# B&R Automation Studio project MotionTestBenchMaster (part 13)

#### ETHIP_COM.st - ETHIP COM Code
```iecst
(************************************************************************************************************************)
(* COPYRIGHT -- Sidel S.p.a.                                                                                            *)
(************************************************************************************************************************)
(* Library:				ETHIP_COM																						*)
(* Author:				Andrea.Cortesi																					*)
(* Site:				Sidel - Parma - Product Care IO																	*)
(* Created:				August 26, 2015																					*)
(* Description:			This Library manage a communication based on ethernet IP Protocol between plc B&R configurated	*)
(*						like a SLAVE and another plc configurated like a MASTER. Connection is openinig only if partner	*)
(*						give positive response at comand ping. In case of timeout connection (5000 ms is default value)	*)
(*						the library close connection, try again to ping partner and if there is no answer generate fault*)
(*						communication. Fault is generate also if there is an error inside Data Object configuration.	*)
(* Restriction:			Call in Fast Task at 30 ms or less.Only one connection can be activated because plc B&R in SLAVE*)
(*						Plc B&R can not be SLAVE of two MASTER at same time!!! Is not possible open two connections like*)
(*						SLAVE concurrently on the same IFx eth port. However is possible open two connections like SLAVE*)
(*						Sconcurrently on two different eth port (ex:IF2 and IF3) with two different IP address class	*)
(* Important Note:		This library open/close connection (with memory release) also in case of program download made	*)
(*						in Copy Mode or Overload Mode.For correct management of Overload Mode is necessaary call istance*)
(*						of ETHIP library with Enable at FALSE inside Exit Transiction of function block in which ETHIP	*)
(*						library istance is called.																		*)
(*----------------------------------------------------------------------------------------------------------------------*)
(* Version History:		v.4.00.0 Date 2015-09-12  Andrea.Cortesi														*)
(* Version History:		v.4.00.1 Date 2017-08-20  Roberto.Bonato														*)
(*																														*)
(*----------------------------------------------------------------------------------------------------------------------*)
(* Development Tool:	B&R Automation Studio V3.0.90.27 SP09															*)
(* Compiler GCC:		V2.95.3; V4.1.1; V4.1.2																			*)
(*----------------------------------------------------------------------------------------------------------------------*)
(* Dependencies:		AsEthIP,AsICMP,AsString,Runtime,Standard														*)
(************************************************************************************************************************)

FUNCTION_BLOCK ETHIP_COM
   (* PING Partner before Communication Initialisation *)
	IF (Enable AND NOT(Ping_Ok) AND NOT(Error)) THEN
		PING_Partner.enable		:= TRUE;
		PING_Partner.pHost		:= ADR(IP_Address_Partner);
		PING_Partner.timeout	:= 500;
		PING_Partner();

		Step_Msg_Active      := 'ETHIP PING';
		Status               := PING_Partner.status;
		ETHIP_COM_Error;	(* Call action ETHIP_COM_Error *)

		CASE PING_Partner.status OF
			0:		(* No Error *)
				Ping_Ok	:= TRUE;

			32750,	(* No response sent by station within the specified timeout *)
			32751,	(* The specified IP address (SG4: name also) could not be resolved *)
			32752,	(* Resource problem in system. Could not create new sockets *)
			65535:	(* No Error - Function block still operating, continue calling *)
				Ping_Ok	:= FALSE;
			ELSE	(* Error not management *)
				Ping_Ok	:= FALSE;
		END_CASE
	END_IF

	(* ETHIP Communication Initialisation *)
	IF ComInit THEN	(* If the communication initialisation is requested then... *)
		ETHIP_Init.enable	:= TRUE;				(* Enabled *)
		ETHIP_Init.pconfig	:= Config_DataObject;	(* Name of the "communication configuration" data object *)
		ETHIP_Init();								(* Call of the "EIPInit" function *)

		Handle_Init			:= ETHIP_Init.handle;	(* The handle returned by the EIPInit Function and is reused by the EIPCyclic AND EIPExit functions *)

		Step_Msg_Active		:= 'ETHIP INIT';
		Status				:= ETHIP_Init.status;
		ETHIP_COM_Error;							(* Call action ETHIP_COM_Error *)

		(* ETHIP Status Init *)
		CASE ETHIP_Init.status OF
			0:		(* No Error *)
				ComInit		:= FALSE;		(* Reset the communication init request *)
				ComStart	:= TRUE;		(* Set the communication activation request *)

			32051,	(* Out of memory. The library cannot be executed *)
			32052,	(* Configuration data object error *)
			32053,	(* Illegal input parameters connected to the FBK. *)
			32054:	(* The Ethernet interface doesn't exist or returns an error. Check the #OWNINTERFACE entry in the configuration data object.*)
				ComInit		:= FALSE;		(* Reset the communication init request *)
				ComStart	:= FALSE;		(* Reset the communication activation request *)
				ComExit		:= TRUE;		(* Set the communication exit request *)

			65534:	(* The FBK was called with enable = 0.*)

			65535:	(* No Error - Function block still operating, continue calling *)

			ELSE	(* Error not management *)
				ComInit		:= FALSE;		(* Reset the communication init request *)
				ComStart	:= FALSE;		(* Reset the communication activation request *)
				ComExit		:= FALSE;		(* Reset the communication exit request *)
		END_CASE
	END_IF

	(* ETHIP Communication Cyclic *)
	IF ComStart THEN		(* If communication activation is requested then... *)
		ETHIP_Cyclic.enable	:= TRUE;		(* Enabled *)
		ETHIP_Cyclic.handle	:= Handle_Init;	(* Handle received from the EIPInit function *)
		ETHIP_Cyclic();						(* Call of the "EIPcyclic" function *)

		Step_Msg_Active		:= 'ETHIP CYCLIC';
		Status				:= ETHIP_Cyclic.status;
		ETHIP_COM_Error;					(* Call action ETHIP_COM_Error *)
	END_IF

	(* ETHIP Status Cyclic *)
	CASE ETHIP_Cyclic.status OF
		0:		(* No Error *)

		32051,	(* Out of memory. The library cannot be executed *)
		32052,	(* Configuration data object error *)
		32053,	(* Illegal input parameters connected to the FBK. *)
		32054:	(* The Ethernet interface doesn't exist or returns an error. Check the #OWNINTERFACE entry in the configuration data object.*)
			ComStart	:= FALSE;		(* Reset the communication activation request *)
			ComExit		:= TRUE;		(* Set the communication exit request *)

		65534:	(* The FBK was called with enable = 0.*)

		65535:	(* No Error - Function block still operating, continue calling *)

		ELSE	(* Error not management *)
			ComInit		:= FALSE;	(* Reset the Communication init request *)
			ComStart	:= FALSE;	(* Reset the communication activation request *)
			ComExit		:= FALSE;	(* Reset the communication exit request *)
	END_CASE

	(* Force ETHIP Communication Exit if Enable Not Active *)
	IF (NOT(Enable) AND (ComStart OR ComInit)) THEN
		ComInit		:= FALSE;	(* Reset the communication init request *)
		ComStart	:= FALSE;	(* Reset the communication activation request *)
		ComExit		:= TRUE;	(* Set the communication exit request *)
	END_IF

	(* ETHIP Communication Exit *)
	IF ComExit THEN	(* If communication exit is requested then... *)
		ComInit		:= FALSE;		(* Reset the communication init request *)
		ComStart	:= FALSE;		(* Reset the communication activation request *)

		ETHIP_Exit.enable	:= TRUE;		(* Enabled *)
		ETHIP_Exit.handle	:= Handle_Init;	(* Handle received from the EIPInit function *)
		ETHIP_Exit();						(* Call of the "EIPExit" function *)

		Step_Msg_Active		:= 'ETHIP EXIT';
		Status				:= ETHIP_Exit.status;
		ETHIP_COM_Error;					(* Call action ETHIP_COM_Error *)
	END_IF

	(* ETHIP Status Exit *)
	CASE ETHIP_Exit.status OF
		0:		(* No Error *)

		32051,	(* Out of memory. The library cannot be executed *)
		32052,	(* Configuration data object error *)
		32053,	(* Illegal input parameters connected to the FBK. *)
		32054:	(* The Ethernet interface doesn't exist or returns an error. Check the #OWNINTERFACE entry in the configuration data object.*)
			ComInit		:= FALSE;	(* Reset the communication init request *)
			ComStart	:= FALSE;	(* Reset the communication activation request *)
			ComExit		:= FALSE;	(* Reset the communication exit request *)

		65534:	(* The FBK was called with enable = 0. *)

		65535:	(* No Error - Function block still operating, continue calling *)

		ELSE	(* Error not management *)
			ComInit		:= FALSE;	(* Reset the communication init request *)
			ComStart	:= FALSE;	(* Reset the communication activation request *)
			ComExit		:= FALSE;	(* Reset the communication exit request *)
	END_CASE

	// Check if ETHIP Communication Exit is Ended
	IF (ComExit AND (ETHIP_Exit.status = 0)) THEN
		ComInit		:= FALSE;		(* Reset the communication init request *)
		ComStart	:= FALSE;		(* Reset the communication activation request *)
		ComExit		:= FALSE;		(* Reset the communication exit request *)
	END_IF

	// Check Presence Status Error in ETHIP Init and ETHIP Cyclic
	IF ((ETHIP_Init.status = 0) OR (ETHIP_Init.status = 65335)) AND ((ETHIP_Cyclic.status = 0) OR (ETHIP_Cyclic.status = 65335)) THEN
		Error_Internal	:= FALSE;	(* Reset Error in ETHIP function *)
	ELSE
		IF Ping_Ok THEN
			Error_Internal	:= TRUE;	(* Set Error in ETHIP function *)
		ELSE
			Error_Internal	:= FALSE;	(* Reset Error in ETHIP function *)
		END_IF
	END_IF

	// Set Communication Exit if Ping Not Ok or Fault Communication
	IF (ComStart AND (EDGEPOS(Error) OR EDGENEG(Ping_Ok))) THEN
		IF ConnectionAttempt > 10 THEN
			ComInit		:= FALSE;		(* Reset the communication init request *)
			ComStart	:= FALSE;		(* Reset the communication activation request *)
			ComExit		:= TRUE;		(* Set the communication exit request *)
			ConnectionAttempt := 0;
		ELSE
			ConnectionAttempt	:= ConnectionAttempt + 1;
			Error := FALSE;
		END_IF
	ELSIF (ComStart AND EDGE(Alive_Bit_From_Partner)) THEN
		ConnectionAttempt := 0;
	END_IF

	// Initializatin Communication
	IF (Enable AND NOT(ComInit) AND NOT(ComStart) AND NOT(ComExit) AND Ping_Ok AND NOT(Error)) THEN
		ComInit		:= TRUE;		(* Set the communication init request *)
		ComStart	:= FALSE;		(* Reset the communication activation request *)
		ComExit		:= FALSE;		(* Reset the communication exit request *)
	END_IF

	// Check TimeOut Value
	IF (TimeOut_Value = 0) THEN
		TimeOut_Value	:= 5000;
	ELSIF (TimeOut_Value < 3000) THEN
		TimeOut_Value	:= 3000;
	END_IF

	// Check Alive Bit Receive from Partner
	IF Enable THEN
		Timer_CommTimeOut(
		IN	:= NOT EDGE(Alive_Bit_From_Partner) AND Timer_StartComDelay.Q,
		PT	:= UINT_TO_TIME(TimeOut_Value)
		);

		Timer_StartComDelay(
		IN	:= TRUE,
		PT	:= UINT_TO_TIME(TimeOut_Value)
		);
	ELSE
		Timer_CommTimeOut(
		IN	:= FALSE,
		PT	:= UINT_TO_TIME(TimeOut_Value)
		);

		Timer_StartComDelay(
		IN	:= FALSE,
		PT	:= UINT_TO_TIME(TimeOut_Value)
		);
	END_IF

	// TimeOut Error Communication
	IF ((NOT(Ping_Ok) AND Timer_CommTimeOut.Q) OR Error_Internal) THEN
		Timer_CommTimeOut.IN	:= FALSE;
		Timer_StartComDelay.IN	:= FALSE;
		Error					:= TRUE;
	END_IF

	// Try again to Ping Partner in case of TimeOut Error Communication
	IF (Ping_Ok AND Timer_CommTimeOut.Q AND NOT(Error)) THEN
		Timer_CommTimeOut.IN	:= FALSE;
		Timer_StartComDelay.IN	:= FALSE;
		Ping_Ok					:= FALSE;
	END_IF

	// Re-initial Communication in CASE OF ERROR
	IF Error THEN
		IF Reset THEN
			Timer_CommTimeOut.IN	:= FALSE;
			Timer_StartComDelay.IN	:= FALSE;
			Error					:= FALSE;
			Ping_Ok					:= FALSE;

			// Reset Buffer and Status
			Buffer_Status_Index		:= 0;
			Status_Old				:= 0;
			Step_Msg_Active_Old		:= '';
			Status_String			:= '';
			memset(ADR(Buffer_Status), 0, SIZEOF(Buffer_Status));

			Step_Msg_Active			:= 'ETHIP RESET';
			Status					:= 55150;	(* Reset Allarm Communication Library *)
			ETHIP_COM_Error;					(* Call action ETHIP_COM_Error *)
		END_IF
	END_IF

	// Call timer
	Timer_CommTimeOut();
	Timer_StartComDelay();
END_FUNCTION_BLOCK
```

#### ETHIP_COM_Error.st - ETHIP COM Error
```iecst
(********************************************************************
 * COPYRIGHT --  Sidel S.p.a.
 ********************************************************************
 * Program: ETHIP_COM
 * File: ETHIP_COM_Error.st
 * Author: Andrea.Cortesi
 * Created: August 26, 2015
 ********************************************************************
 * Implementation of program ETHIP_COM
 ********************************************************************)

ACTION ETHIP_COM_Error:

	CASE Status OF

		0    : Msg_Error := 'No Error';
		55100: Msg_Error := 'Error Enable Library File_CSV Not Coerent';
		55101: Msg_Error := 'Error File CSV Actual is Empty (size zero)';
		55102: Msg_Error := 'Error File CSV Old is Empty (size zero)';
		55103: Msg_Error := 'Force Exit from Sequencer Library FILE_CSV';
		55104: Msg_Error := 'File CSV Saved - No Error';
		55105: Msg_Error := 'File CSV Loaded - No Error';
		55106: Msg_Error := 'Error Step Sequencer in Library FILE_CSV';
		55150: Msg_Error := 'Reset Error Communication Library';
		9999 : Msg_Error := 'FUNCTION NOT implemented';
		20700: Msg_Error := 'Invalid path; check the path specification (AND length OF path)';
		20701: Msg_Error := 'The specified data length is too small';
		20702: Msg_Error := 'No more file handles available';
		20703: Msg_Error := 'Code error (system error)';
		20704: Msg_Error := 'Invalid TYPE';
		20705: Msg_Error := 'File already exists';
		20706: Msg_Error := 'ACCESS NOT possible using the desired mode';
		20707: Msg_Error := 'FiERR_MODE  Illegal mode';
		20708: Msg_Error := 'File does NOT exist';
		20709: Msg_Error := 'Illegal file device (e.g. not initialized "CPU -> Properties -> File Devices")';
		20710: Msg_Error := 'NOT enough memory FOR file with new write data';
		20711: Msg_Error := 'Invalid file offset';
		20712: Msg_Error := 'File NOT allowed';
		20713: Msg_Error := 'NOT enough memory (DRAM) available TO copy file';
		20714: Msg_Error := 'General error in FileOpen';
		20715: Msg_Error := 'General error in FileClose';
		20716: Msg_Error := 'General error in FileRead';
		20717: Msg_Error := 'General error in FileWrite';
		20718: Msg_Error := 'General error in Ioctl';
		20719: Msg_Error := 'The specified POINTER is invalid (NULL)';
		20720: Msg_Error := 'Error in the FileIO manager';
		20721: Msg_Error := 'File NOT open';
		20722: Msg_Error := 'Invalid directory';
		20723: Msg_Error := 'Directory does NOT exist';
		20724: Msg_Error := 'Directory NOT empty';
		20725: Msg_Error := 'Directory already exists';
		20726: Msg_Error := 'Error retrieving memory information';
		20727: Msg_Error := 'NOT enough memory available on the target device (FileCopy)';
		20728: Msg_Error := 'Idents directory no longer available. Close open directories (or free up memory)';
		20729: Msg_Error := 'Invalid parameter output';
		20730: Msg_Error := 'Directory already exists';
		20731: Msg_Error := 'The specified handle is invalid';
		20732: Msg_Error := 'Another IP address has already been defined FOR a host name';
		20796: Msg_Error := 'Could NOT initialize library';
		20797: Msg_Error := 'Error in device driver';
		20798: Msg_Error := 'Error in device manager';
		20799: Msg_Error := 'System error.General system fault';
		32051: Msg_Error := 'Out of memory. The library cannot be executed';
		32052: Msg_Error := 'Configuration data object error';
		32053: Msg_Error := 'Illegal input parameters connected to the Function block';
		32054: Msg_Error := 'Ethernet interface not exist or in error.Check #OWNINTERFACE data object';
		32750: Msg_Error := 'No response sent by station within the specified timeout';
		32751: Msg_Error := 'The specified IP address (SG4: name also) could not be resolved';
		32752: Msg_Error := 'Resource problem in system. Could not create new sockets';
		32799: Msg_Error := 'System error';
		65534: Msg_Error := 'Function block was called with enable at FALSE';
		65535: Msg_Error := 'Function block continue calling';

	ELSE

			   Msg_Error := 'Error not management';

	END_CASE

	// Buffer Status for Diagnostic
	IF ((Status <> Status_Old) OR ((strcmp(ADR(Step_Msg_Active),ADR(Step_Msg_Active_Old))) <> 0)) AND (Buffer_Status_Index < Buffer_Status_MaxLimit) THEN
		itoa(UINT_TO_DINT(Status),ADR(Status_String));
		Status_String                      := CONCAT(Status_String,': ');
		Status_String                      := CONCAT(Status_String,Step_Msg_Active);
		Status_String                      := CONCAT(Status_String,': ');
		Buffer_Status[Buffer_Status_Index] := CONCAT(Status_String,Msg_Error);
		Buffer_Status_Index                := (Buffer_Status_Index + 1);

		// Update Status Old if Change
		IF (Status <> Status_Old) THEN
			Status_Old := Status;
		END_IF
		// Update Step Msg active Old if Changed
		IF ((strcmp(ADR(Step_Msg_Active),ADR(Step_Msg_Active_Old))) <> 0) THEN
		    Step_Msg_Active_Old := Step_Msg_Active;
		END_IF
		// Reset Buffer Status if is Fu
		IF (Buffer_Status_Index = Buffer_Status_MaxLimit) THEN
		    // Reset Buffer and Status
		    Buffer_Status_Index      := 0;
			Status_Old               := 0;
			Step_Msg_Active_Old      := '';
		    memset(ADR(Buffer_Status),0,SIZEOF(Buffer_Status));
		END_IF

	END_IF

END_ACTION
```

### Package Logical/00_AID/Libraries/System_Libraries - Global libraries

### Global_Constants.var - Global constants
```iecst
(*PROJECT TYPE*)
VAR CONSTANT
	CST_AID_ProjectMachine : USINT := 1;
	CST_AID_ProjectSkid : USINT := 2;
END_VAR
(*COP*)
VAR CONSTANT
	CST_COP_RcpMax : USINT := 10;
	CST_COP_PhaseMaxNr : USINT := 150;
END_VAR
(*FMC*)
VAR CONSTANT
	CST_FmcModeIdle : USINT := 0; (*Filling Master Card Mode IDLE*)
	CST_FmcModeOperation : USINT := 1; (*Filling Master Card Mode OPERATION*)
	CST_FmcModeCipRinse : USINT := 2; (*Filling Master Card Mode CIP/RINSE*)
END_VAR
(*CONFIGURATION*)
VAR CONSTANT
	MIN_CFG_PSx : UINT := 200;
	MAX_CFG_PSx : UINT := 299; (*v1.7.4*)
	MIN_CFG_LSx : UINT := 200;
	MAX_CFG_LSx : UINT := 299;
	MIN_CFG_HSx : UINT := 200; (*V4.A.A.1.6.12*)
	MAX_CFG_HSx : UINT := 299; (*V4.A.A.1.6.12*)
	MIN_CFG_FSx : UINT := 200;
	MAX_CFG_FSx : UINT := 299;
	MIN_CFG_GSx : UINT := 200;
	MAX_CFG_GSx : UINT := 299;
	MIN_CFG_QSx : UINT := 200; (*v1.7.4*)
	MAX_CFG_QSx : UINT := 299; (*v1.7.4*)
	MIN_CFG_CTx : UINT := 200;
	MAX_CFG_CTx : UINT := 300;
	MIN_CFG_QTx : UINT := 200;
	MAX_CFG_QTx : UINT := 300;
	MIN_CFG_FTx : UINT := 200;
	MAX_CFG_FTx : UINT := 310;
	MIN_CFG_TTx : UINT := 200;
	MAX_CFG_TTx : UINT := 300;
	MIN_CFG_TSx : UINT := 200;
	MAX_CFG_TSx : UINT := 300;
	MIN_CFG_PTx : UINT := 200;
	MAX_CFG_PTx : UINT := 310;
	MIN_CFG_LTx : UINT := 200;
	MAX_CFG_LTx : UINT := 210;
	MIN_CFG_RVx : UINT := 200;
	MAX_CFG_RVx : UINT := 299;
	MIN_CFG_PID_PPx : UINT := 200;
	MAX_CFG_PID_PPx : UINT := 220; (*V4.A.A.1.7.1*)
	MIN_CFG_PID_RVx : UINT := 200;
	MAX_CFG_PID_RVx : UINT := 220;
	MIN_CFG_PID_RMx : UINT := 200;
	MAX_CFG_PID_RMx : UINT := 210;
	MIN_CFG_RMx : UINT := 200;
	MAX_CFG_RMx : UINT := 210;
	MIN_CFG_MMx : UINT := 200;
	MAX_CFG_MMx : UINT := 299;
	MIN_CFG_PPx : UINT := 200;
	MAX_CFG_PPx : UINT := 299;
	MIN_CFG_AVx : UINT := 200;
	MAX_CFG_AVx : UINT := 299;
	MIN_CFG_HVx : UINT := 200; (*V4.A.A.1.6.12*)
	MAX_CFG_HVx : UINT := 299; (*V4.A.A.1.6.12*)
	MIN_CFG_EVx : UINT := 200; (*v1.7.4*)
	MAX_CFG_EVx : UINT := 299; (*v1.7.4*)
	MIN_CFG_VFD_MMx : UINT := 200;
	MAX_CFG_VFD_MMx : UINT := 210;
	MIN_CFG_VFD_PPx : UINT := 200;
	MAX_CFG_VFD_PPx : UINT := 220;
	MIN_SS3P_CFG : UINT := 0;
	MAX_SS3P_CFG : UINT := 20;
	MIN_SS2P_CFG : UINT := 0;
	MAX_SS2P_CFG : UINT := 20;
	MAX_SS2P_DMC : UINT := 3;
	MIN_PB_CFG : UINT := 0;
	MAX_PB_CFG : UINT := 20;
	MIN_CFG_LOTO_Step : UINT := 0;
	MAX_CFG_LOTO_Step : UINT := 19;
	MIN_CFG_LOTO_Condition : UINT := 0;
	MAX_CFG_LOTO_Condition : UINT := 31;
	MIN_CFG_TPM_Bar : UINT := 0;
	MAX_CFG_TPM_Bar : UINT := 24;
	MIN_CmdBar_PB : UINT := 1;
	MAX_CmdBar_PB : UINT := 25;
	MIN_CFG_SafetyZone : UINT := 1;
	MAX_CFG_SafetyZone : UINT := 22;
	MIN_CFG_SafetyDoor : UINT := 1;
	MAX_CFG_SafetyDoor : UINT := 8;
	MIN_CFG_SafetyDoorCabinet : UINT := 1;
	MAX_CFG_SafetyDoorCabinet : UINT := 5;
	MIN_CFG_SafetyEmergency : UINT := 1;
	MAX_CFG_SafetyEmergency : UINT := 11;
	MIN_CFG_SafetyJog : UINT := 0;
	MAX_CFG_SafetyJog : UINT := 22;
	MAX_CFG_DoorConfiguration : UINT := 40;
	MAX_CFG_JogConfiguration : UINT := 30;
	MAX_CFG_EmergencyConfiguration : UINT := 30;
END_VAR
(*CONFIGURATION C Family 1.7.2*)
VAR CONSTANT
	MIN_CFG_PSC : UINT := 200;
	MAX_CFG_PSC : UINT := 210;
	MIN_CFG_HSC : UINT := 200;
	MAX_CFG_HSC : UINT := 209;
	MIN_CFG_LSC : UINT := 200;
	MAX_CFG_LSC : UINT := 209;
	MIN_CFG_FSC : UINT := 200;
	MAX_CFG_FSC : UINT := 299;
	MIN_CFG_GSC : UINT := 200;
	MAX_CFG_GSC : UINT := 209;
	MIN_CFG_CTC : UINT := 200;
	MAX_CFG_CTC : UINT := 209;
	MIN_CFG_QTC : UINT := 200;
	MAX_CFG_QTC : UINT := 209;
	MIN_CFG_FTC : UINT := 200;
	MAX_CFG_FTC : UINT := 209;
	MIN_CFG_TTC : UINT := 200;
	MAX_CFG_TTC : UINT := 209;
	MIN_CFG_TSC : UINT := 200;
	MAX_CFG_TSC : UINT := 209;
	MIN_CFG_PTC : UINT := 200;
	MAX_CFG_PTC : UINT := 209;
	MIN_CFG_LTC : UINT := 200;
	MAX_CFG_LTC : UINT := 209;
	MIN_CFG_RVC : UINT := 200;
	MAX_CFG_RVC : UINT := 209;
	MIN_CFG_PID_PPC : UINT := 200;
	MIN_CFG_PID_RVC : UINT := 200;
	MAX_CFG_PID_RVC : UINT := 209;
	MIN_CFG_PID_RMC : UINT := 200;
	MAX_CFG_PID_RMC : UINT := 209;
	MIN_CFG_RMC : UINT := 200;
	MAX_CFG_RMC : UINT := 209;
	MIN_CFG_MMC : UINT := 200;
	MAX_CFG_MMC : UINT := 209;
	MIN_CFG_PPC : UINT := 200;
	MAX_CFG_PPC : UINT := 209;
	MIN_CFG_AVC : UINT := 100;
	MAX_CFG_AVC : UINT := 209;
	MIN_CFG_HVC : UINT := 200;
	MAX_CFG_HVC : UINT := 209;
	MIN_CFG_VFD_MMC : UINT := 200;
	MAX_CFG_VFD_MMC : UINT := 209;
	MIN_CFG_VFD_PPC : UINT := 200;
	MAX_CFG_VFD_PPC : UINT := 209;
END_VAR
(*Vfd Node*)
VAR CONSTANT
	MIN_CFG_VfdNode : UINT := 220; (*V4.A.A.1.7.6*)
	MAX_CFG_VfdNode : UINT := 240; (*V4.A.A.1.7.6*)
END_VAR
(*Sequencer*)
VAR CONSTANT
	MAX_STEP_CFG : UINT := 201;
	MAX_JUMP_CFG : UINT := 30;
END_VAR
(*Jog Speed *)
VAR CONSTANT
	CST_JogMinimumSpeed : REAL := 500.0;
	CST_JogMaximumSpeed : REAL := 3000.0;
END_VAR
(*Filler Shift Constant*)
VAR CONSTANT
	CST_ShiftDimensionCombi : UINT := 1000; (*Machine Shift Array*)
	CST_ShiftDimension : UINT := 1000; (*Machine Shift Array*)
END_VAR
```

### Command_Bar_Constants.var - Global constants
```iecst
(*COMMAND BAR PB*)
VAR CONSTANT
	PB_MixerProcessStart : USINT := 1;
	PB_FillerProcessStart : USINT := 2;
	PB_FillerStartStop : USINT := 4;
	PB_SeamerStartStop : USINT := 5;
	PB_FillerDoorUnlock : USINT := 11;
	PB_SeamerDoorUnlock : USINT := 14;
	PB_ContainerBlock1 : USINT := 15;
	PB_ContainerRelease1 : USINT := 16;
	PB_ContainerBlock2 : USINT := 17;
	PB_ContainerRelease2 : USINT := 18;
	PB_FillerLabellerCoupling : USINT := 19;
	PB_FillerBlowerCoupling : USINT := 20;
	PB_FillerSeamerCoupled : USINT := 21;
	PB_FillerActisCoupled : USINT := 22; (*V4.A.A.1.6.13*)
END_VAR
```

### Counter_Constants.var - Global constants
```iecst
(*Machine Counters*)
VAR CONSTANT
	FillerLaps : USINT := 0;
	ClosingUnit1Laps : USINT := 1;
	ClosingUnit2Laps : USINT := 2;
	RinserLaps : USINT := 3;
	FlaworDoserLaps : USINT := 4;
	PulpDoserLaps : USINT := 5;
	PowerOn : USINT := 6;
	RotatingTime : USINT := 7;
	PowerOnTime : USINT := 8;
END_VAR
(*Containers Counters*)
VAR CONSTANT
	FillingFault : USINT := 0;
	FillingBurst : USINT := 1;
	ClosingUnit1Fault : USINT := 2;
	ClosingUnit2Fault : USINT := 3;
	RinsingFault : USINT := 4;
	PulpDoserFault : USINT := 5;
	FlaworDoserFault : USINT := 6;
	BurstEjected : USINT := 7;
	ManualEjected : USINT := 8;
	LowFillingEjected : USINT := 9;
	NotFilledEjected : USINT := 10;
	ContainersEntered : USINT := 11;
	ContainersProduced : USINT := 12;
	EjectionBySIS : USINT := 13;
	BottleProduceToCvo : USINT := 14;
	Spare : USINT := 15;
END_VAR
(*Process Counters*)
VAR CONSTANT
	FillerProduction : USINT := 0;
	ClosingUnit1Production : USINT := 1;
	ClosingUnit2Production : USINT := 2;
	RinserProduction : USINT := 3;
	PulpDoserProduction : USINT := 4;
	FlaworDoserProduction : USINT := 5;
	Cop : USINT := 6;
	FillerCip : USINT := 7;
	ClosingUnit1Cip : USINT := 8;
	ClosingUnit2Cip : USINT := 9;
	RinserCip : USINT := 10;
	PulpDoserCip : USINT := 11;
	FlaworDoserCip : USINT := 12;
END_VAR
(*ECO Counters*)
VAR CONSTANT
	Power : USINT := 0;
	Air : USINT := 1;
	GeneralCO2 : USINT := 2;
	ClosingUnitCO2 : USINT := 3;
	N2 : USINT := 4;
	ProcessWater : USINT := 5;
	CopWater : USINT := 6;
	BottomBottleCoolingWater : USINT := 7;
	Product : USINT := 8;
	Steam : USINT := 9;
	FoodSteam : USINT := 10;
	ProductWater : USINT := 11;
	Syrup : USINT := 12; (*V4.A.A.1.6.14k*)
END_VAR
```

### ITC_Constants.var - Global constants
```iecst
(*Coupled Machine*)
VAR CONSTANT
	CST_ITC_BLR : USINT := 11; (*Blower*)
	CST_ITC_LBR : USINT := 12; (*Labeller*)
	CST_ITC_SMF : USINT := 13; (*Seamer Ferrum*)
	CST_ITC_ACTIS : USINT := 14; (*Actis*)
	CST_ITC_PULPDOSER : USINT := 15; (*Pulp Doser*)
	CST_ITC_CLOSINGUNIT : USINT := 16; (*Closing unit*)
	CST_ITC_FLAVORDOSER : USINT := 17; (*Flavor Doser//1.63*)
END_VAR
(*Sidel Process*)
VAR CONSTANT
	CST_ITC_SKD_FLR : USINT := 21; (*Skid/Filler*)
	CST_ITC_COREBLEND : USINT := 22; (*Coreblend*)
END_VAR
(*External Process*)
VAR CONSTANT
	CST_ITC_MXR : USINT := 31; (*Mixer*)
	CST_ITC_CARBO : USINT := 32; (*Carbo*)
	CST_ITC_PRD : USINT := 33; (*Product Room*)
	CST_ITC_BBT : USINT := 34; (*BBT*)
	CST_ITC_ASEPTICTANK : USINT := 35; (*Aseptic Tank*)
END_VAR
(*Product treatments (41-49 RESERVED SKID)*)
(*Hygiene*)
VAR CONSTANT
	CST_ITC_CIP : USINT := 51; (*CIP Room*)
	CST_ITC_COP : USINT := 52; (*COP*)
	CST_ITC_WHITEROOM : USINT := 53; (*White room*)
END_VAR
(*External equipments*)
VAR CONSTANT
	CST_ITC_CVI : USINT := 61; (*Inlet Conveyor*)
	CST_ITC_CVO : USINT := 62; (*Outlet Conveyor*)
	CST_ITC_FCI : USINT := 63; (*Filler Container Inspector*)
	CST_ITC_VBC : USINT := 64; (*Vacuum Barrier Company*)
	CST_ITC_CFD : USINT := 65; (*Cap Feeder*)
	CST_ITC_CFD2 : USINT := 66; (*Cap Feeder 2*)
	CST_ITC_CDR : USINT := 67; (*Coder*)
	CST_ITC_LDF : USINT := 68; (*Lid feeder*)
	CST_ITC_UVL : USINT := 69; (*UV Lamp Caps treatment v1.4*)
END_VAR
(*External equipments 2*)
VAR CONSTANT
	CST_ITC_SIKO : USINT := 81; (*Arol Siko Multibody V4.A.A.1.6.12*)
	CST_ITC_WTT : USINT := 82; (*Water system Water treatment Rinser V4.A.A.1.6.12*)
	CST_ITC_CDS : USINT := 83; (*Cap Dis   V4.A.A.1.7.0*)
	CST_ITC_PST : USINT := 85; (*v999hema*)
END_VAR
(*Data*)
VAR CONSTANT
	CST_ITC_SCC : USINT := 71; (*Signals Customer Concentrator*)
	CST_ITC_DATA : USINT := 72; (*Data Acquisition*)
	CST_ITC_PCO : USINT := 73; (*Product change over*)
END_VAR
(*Communication Status*)
VAR CONSTANT
	CST_CommStatus_NotPresent : USINT := 0;
	CST_CommStatus_NotConnected : USINT := 1;
	CST_CommStatus_Connecting : USINT := 2;
	CST_CommStatus_Connected : USINT := 3;
END_VAR
```

### PB_Constants.var - Push buttons constants
```iecst
(*General*)
VAR CONSTANT
	PB_CmdStop : USINT := 0;
	PB_CmdStart : USINT := 1;
	PB_CmdSkip : USINT := 2;
	PB_CmdPause : USINT := 3;
	PB_CmdAbort : USINT := 4;
END_VAR
(*CAP*)
VAR CONSTANT
	PB_GeasingCmdStart : USINT := 2;
	PB_CAP_HeadChartDataReset : USINT := 4; (*V4.A.A.1.6.11*)
	PB_CAP_RecipeDataRestore : USINT := 5; (*V4.A.A.1.6.11*)
	PB_CAP_DataStore : USINT := 6; (*V4.A.A.1.6.11*)
	PB_CAP_HeadDataRestore : USINT := 7; (*V4.A.A.1.6.11*)
	PB_CAP_HeadJogBackward : USINT := 8; (*V4.A.A.1.6.11*)
	PB_CAP_HeadJogForward : USINT := 9; (*V4.A.A.1.6.11*)
	PB_CAP_BufferAdjustReduce : USINT := 12; (*V4.A.A.1.6.11*)
	PB_CAP_BufferAdjustExpand : USINT := 13; (*V4.A.A.1.6.11*)
END_VAR
(*CSR*)
VAR CONSTANT
	PB_CSR_ConveyorCalibration : USINT := 1;
	PB_CSR_ConveyorParDownload : USINT := 6;
	PB_CSR_ConveyorParUpload : USINT := 7;
	PB_CSR_ConveyorGuideCalibration : USINT := 8;
	PB_CSR_ConveyorGuideParDownload : USINT := 9;
	PB_CSR_ConveyorGuideParUpload : USINT := 2;
	PB_CSR_PositionOffset : USINT := 3;
	PB_CSR_PositionOffsetDec : USINT := 4;
	PB_CSR_PositionOffsetInc : USINT := 13;
	PB_CSR_PositionGuideOffset : USINT := 14;
	PB_CSR_PositionGuideOffsetDec : USINT := 17;
	PB_CSR_PositionGuideOffsetInc : USINT := 18;
	PB_CSR_Down : USINT := 16;
	PB_CSR_LiftConfirm : USINT := 5;
	PB_CSR_SkfInit : USINT := 10; (*SKF Control Unit -System Initialization*)
	PB_CSR_SkfAcquireLowPos : USINT := 11; (*SKF Control Unit -Lowest Position Permitted*)
	PB_CSR_SkfAcquireHighPos : USINT := 12; (*SKF Control Unit -Highest Position Permitted*)
	PB_CSR_Up : USINT := 15;
	PB_CSR_Down : USINT := 16;
	PB_CSR_CrownerPositioning : USINT := 19; (*V4.A.A.1.7.0*)
	PB_CSR_CapperPositioning : USINT := 20; (*V4.A.A.1.7.0*)
END_VAR
(*HMI*)
VAR CONSTANT
	PB_PAR_Initialization : USINT := 0;
	PB_CFG_SavePao : USINT := 1;
	PB_CFG_LoadPao : USINT := 2;
	PB_CFG_SaveCfg : USINT := 3;
	PB_CFG_LoadCfg : USINT := 4;
	PB_BeaconTest : USINT := 5;
END_VAR
(*MAU*)
VAR CONSTANT
	PB_MAU_MachineLight : USINT := 2;
END_VAR
(*MAU Container Lubrication*)
VAR CONSTANT
	PB_LbCon_Test : USINT := 10;
END_VAR
(*MAU Container Chloride Water Washing*)
VAR CONSTANT
	PB_LbCon_Cmd : USINT := 11;
	PB_LbInt_Cmd : USINT := 12;
END_VAR
(*MAU Lift Lubrification*)
VAR CONSTANT
	PB_LbConExtLift_Cmd : USINT := 13;
END_VAR
(*MAU Dummy Container*)
VAR CONSTANT
	PB_DumCon_FirstHalfPos : USINT := 0;
	PB_DumCon_SecondHalfPos : USINT := 1;
	PB_DumCon_FirstHalfPistonDown : USINT := 2;
	PB_DumCon_SecondHalfPistonDown : USINT := 3;
	PB_DumCon_FirstHalfRotToProd : USINT := 4;
	PB_DumCon_SecondHalfRotToProd : USINT := 5;
	PB_DumCon_FirstHalfRotToCip : USINT := 6;
	PB_DumCon_SecondHalfRotToCip : USINT := 7;
	PB_DumCon_FirstHalfPistonUp : USINT := 8;
	PB_DumCon_SecondHalfPistonUp : USINT := 9;
	PB_DumCon_FirstHalfStartCheck : USINT := 10;
	PB_DumCon_SecondHalfStartCheck : USINT := 11;
END_VAR
(*MAU Greasing*)
VAR CONSTANT
	PB_GrLb_Manual : USINT := 0;
END_VAR
(*MNM*)
VAR CONSTANT
	PB_MNM_AxisHoming : USINT := 2;
	PB_MNM_AxisPositioning : USINT := 3;
	PB_MNM_AxisStepByStep : USINT := 4;
	PB_MNM_AxisInMotionAdjustment : USINT := 5;
	PB_MNM_FootboardPosition : USINT := 6;
	PB_MNM_BrakeRelease : USINT := 7;
	PB_MNM_VelocityTest : USINT := 8;
	PB_MNM_Autotuning : USINT := 9;
	PB_MNM_MotorSetup : USINT := 10;
	PB_MNM_RinserFootboardPosition : USINT := 12; (*V4.A.A.1.7.0*)
END_VAR
(*OPS*)
VAR CONSTANT
	PB_OPS_SaveCfg : USINT := 0;
END_VAR
(*RNS*)
VAR CONSTANT
	PB_RNS_CounterReset : USINT := 5; (*V4.A.A.1.7.0*)
	PB_RNS_PageUp : USINT := 6; (*V4.A.A.1.7.0*)
	PB_RNS_PageDown : USINT := 7; (*V4.A.A.1.7.0*)
END_VAR
(*SFT*)
VAR CONSTANT
	PB_SFT_CounterReset : USINT := 0;
	PB_SFT_SamplingMoldStart : USINT := 1; (*v1.63*)
	PB_SFT_SamplingMoldSelectAll : USINT := 2; (*v1.63*)
	PB_SFT_SamplingMoldReset : USINT := 3; (*v1.63*)
	PB_SFT_SamplingReq : USINT := 10;
	PB_SFT_BurstColorStatusReset : USINT := 11; (*Master nuovo*)
	PB_SFT_BurstCounterReset : USINT := 12;
	PB_SFT_BurstAckowledge : USINT := 13; (*Master nuovo*)
END_VAR
(*TNK*)
VAR CONSTANT
	PB_TNK_ModeEndProd : USINT := 5;
	PB_TNK_CO2_Purge : USINT := 6;
	PB_TNK_Priming : USINT := 7; (*Filling Valves Priming *)
	PB_TNK_StartAutotuning : USINT := 10; (*PPF201 Autotuning Start*)
	PB_TNK_StopAutotuning : USINT := 11; (*PPF201 Autotuning Stop*)
	PB_TNK_SaveAutotuning : USINT := 12; (*PPF201 Autotuning Save New Values*)
	PB_TNK_SamplingReq : USINT := 10;
END_VAR
(*CONTAINER BURST HMI BUTTONS*)
VAR CONSTANT
	PB_BBT_Restore : USINT := 0; (*Master nuovo*)
	PB_BBT_CounterReset : USINT := 1; (*Master nuovo*)
END_VAR

VAR CONSTANT
	PB_CmdDosStop : USINT := 0; (*v999hema*)
	PB_CmdDosStart : USINT := 1;
	PB_CmdDosSkip : USINT := 2;
	PB_CmdDosPause : USINT := 3;
	PB_CmdDosAbort : USINT := 4;
	PB_CmdLiftMotorStop : USINT := 5;
	PB_CmdLiftMotorStart : USINT := 6;
	PB_DOS_Up : USINT := 7;
	PB_DOS_Down : USINT := 8;
END_VAR
```

### SS2P_Constants.var - Selectors switch two positions constants
```iecst
(*General*)
VAR CONSTANT
	SS2P_SelAutoMan : USINT := 0;
	SS2P_SelProduction : USINT := 1;
	SS2P_SelEmptying : USINT := 2;
	SS2P_SelDrain : USINT := 3;
	SS2P_SelCIP : USINT := 4;
END_VAR
(*BTC*)
VAR CONSTANT
	SS2P_BTC_UvLampEnable : USINT := 5;
	SS2P_BTC_WaterCooling : USINT := 6;
END_VAR
(*CAP*)
VAR CONSTANT
	SS2P_CAP_BufferSafety : USINT := 4;
	SS2P_CAP_CapsReleaseSafety : USINT := 5;
	SS2P_CAP_ChannelSafety : USINT := 6;
	SS2P_CAP_InfeedBufferEmptying : USINT := 8;
	SS2P_CAP_CompleteEmptying : USINT := 9;
	SS2P_CAP_GreasingCycle : USINT := 10;
	SS2P_CAP_SizeChangeCmd : USINT := 11;
	SS2P_CAP_EquaRotationCmd : USINT := 12; (*v1.7.4a*)
	SS2P_CAP_StartCalibrationCmd : USINT := 13;
	SS2P_CAP_ZeroEncoderCmd : USINT := 14;
	SS2P_CAP_DataStoreCmd : USINT := 15;
	SS2P_CAP_HRMRotationCmd : USINT := 16; (*v1.7.4a*)
	SS2P_SikoChangeGuideAutoMan : USINT := 17; (*V4.A.A.1.6.12*)
	SS2P_CAP_BufferAdjustManual : USINT := 18; (*V4.A.A.1.6.11*)
	SS2P_CAP_BufferAdjustToTarget : USINT := 19; (*V1.7.4*)
	SS2P_CAP_GreasingCycle_Pump2 : USINT := 20; (*v1.7.5*)
END_VAR
(*CRW*)
VAR CONSTANT
	SS2P_CRW_CrownsReleaseSafety : USINT := 5;
	SS2P_CRW_ChannelSafety : USINT := 6;
	SS2P_CRW_ChannelEmptying : USINT := 8;
END_VAR
(*CO*)
VAR CONSTANT
	SS2P_APCO_ON : USINT := 0;
	SS2P_APCO_PrcChRcp : USINT := 1; (*V4.A.A.1.6.12*)
END_VAR
(*COP*)
VAR CONSTANT
	SS2P_COP_FoamingGun : USINT := 1; (*Foaming in Manual Mode - Present if Cip of Cop*)
	SS2P_COP_Drain : USINT := 2;
	SS2P_COP_CipMode : USINT := 3; (*Cleaning in Auto Mode - Present if Cip of Cop*)
	SS2P_COP_Priming : USINT := 4;
	SS2P_COP_ExtCleaning : USINT := 7;
	SS2P_COP_Satellites : USINT := 9;
	SS2P_COP_DmcManual : USINT := 10; (*V4.A.A.1.7.0*)
	SS2P_COP_WashInProduction : USINT := 11; (*vrmaWIP*)
END_VAR
(*CSR*)
VAR CONSTANT
	SS2P_CSR_ManualTank : USINT := 1;
	SS2P_CSR_ManualCamma : USINT := 2;
	SS2P_CSR_ManualRns : USINT := 3;
	SS2P_CSR_ManualCrw : USINT := 4;
	SS2P_CSR_SectorUnlock : USINT := 5;
	SS2P_CSR_ManualCap : USINT := 6; (*master Nuovo*)
	SS2P_CSR_ConveyorEnable : USINT := 7; (*V4.A.A.1.6.12*)
	SS2P_CSR_ConveyorGuideEnable : USINT := 8; (*V4.A.A.1.6.12*)
	SS2P_CSR_ConveyorGuideSelection : USINT := 9; (*V4.A.A.1.6.12*)
	SS2P_CSR_ConveyorSelection : USINT := 10; (*V4.A.A.1.6.12*)
END_VAR
(*RNS*)
VAR
	SS2P_RNS_InsControl : {REDUND_UNREPLICABLE} USINT := 5; (*V4.A.A.1.7.0*)
	SS2P_RNS_ContControl : {REDUND_UNREPLICABLE} USINT := 6; (*V4.A.A.1.7.0*)
	SS2P_RNS_Bypass : {REDUND_UNREPLICABLE} USINT := 7; (*V4.A.A.1.7.0*)
	SS2P_RNS_EnableCip : {REDUND_UNREPLICABLE} USINT := 8; (*V4.A.A.1.7.0*)
END_VAR
(*HMI*)
VAR CONSTANT
	SS2P_HMI_DeviceEnable : USINT := 0;
	SS2P_HMI_SelEnable : USINT := 1;
	SS2P_HMI_PilotAirUnload : USINT := 2;
END_VAR
(*MAU Container lifting*)
VAR CONSTANT
	SS2P_LftCon_BlowOff : USINT := 3; (*HMI_LftCon_SS2P*)
END_VAR
(*MAU Dummy Containers*)
VAR CONSTANT
	SS2P_DumCon_ManualTest : USINT := 0;
	SS2P_DumCon_DiscargeAir : USINT := 1;
	SS2P_DumCon_ManualMode : USINT := 2;
END_VAR
(*MAU Container Chloride Water Washing*)
VAR CONSTANT
	SS2P_HMI_ChlDioxineEnable : USINT := 1;
	SS2P_HMI_MaxCounter : USINT := 2;
END_VAR
(*MAU White room*)
VAR CONSTANT
	SS2P_WhRoom_Enable : USINT := 1;
END_VAR
(*OPT SS2P*)
VAR CONSTANT
	SS2P_OPT_VbcEnable : USINT := 0;
	SS2P_OPT_FciEnable : USINT := 1;
	SS2P_OPT_CoderEnable : USINT := 2;
	SS2P_OPT_StopForBurstInspection : USINT := 3;
	SS2P_OPT_IntelliChangeOverEnable : USINT := 9;
	SS2P_OPT_CvoSlowDown : USINT := 10;
	SS2P_OPT_FerrumGasEnable : USINT := 15;
	SS2P_OPT_DoubleInletDoubleBlock : USINT := 16;
END_VAR
(*SFT*)
VAR CONSTANT
	SS2P_SFT_StepCounter : USINT := 5;
	SS2P_SFT_BlowerCountingEn : USINT := 6; (*v1.4*)
	SS2P_SFT_BottleEjectorManualTest : USINT := 7; (*v1.63*)
	SS2P_SFT_BlowerSamplingEnable : USINT := 8; (*v1.63*)
	SS2P_SFT_PreformManualLoading : USINT := 9; (*v1.6*)
	SS2P_SFT_SamplingMode : USINT := 10;
	SS2P_SFT_SamplingNoFill : USINT := 11;
	SS2P_SFT_BlowerSamplingEnable : USINT := 8; (*V4.A.A.1.6.12*)
	SS2P_SFT_SamplingNoCap : USINT := 12;
	SS2P_SFT_InletContBlock1_ManTest : USINT := 15;
	SS2P_SFT_InletContBlock2_ManTest : USINT := 16;
END_VAR
(*SMR*)
VAR CONSTANT
	SS2P_SMR_ModeCip : USINT := 0;
	SS2P_SMR_ModeRinse : USINT := 2;
	SS2P_SMR_ModeProd : USINT := 3;
	SS2P_SMR_TestOp1 : USINT := 10;
	SS2P_SMR_RoofOpening : USINT := 11;
	SS2P_SMR_GasManualMode : USINT := 12;
END_VAR
(*TNK*)
VAR CONSTANT
	SS2P_TNK_ModeCIP : USINT := 0;
	SS2P_TNK_ModeDrain : USINT := 1;
	SS2P_TNK_ModeRinse : USINT := 2;
	SS2P_TNK_ModeProdFast : USINT := 3; (*Production Start Up (Heating With Product)*)
	SS2P_TNK_ModeProdStill : USINT := 4;
	SS2P_TNK_ModeProdFlooding : USINT := 5;
	SS2P_TNK_ModeProdFlushing : USINT := 6;
	SS2P_TNK_ModeProdHeatingDB : USINT := 7; (*Heating With Dummy Bottles*)
	SS2P_TNK_ModeProdHeatingWater : USINT := 8; (*Heating With Water*)
	SS2P_TNK_ModeRinseQuick : USINT := 9;
	SS2P_TNK_ModeRinseFast : USINT := 10;
	SS2P_TNK_PrimingTray : USINT := 11; (*Priming Tray In/Out*)
	SS2P_TNK_TanksDrain : USINT := 12; (*Product and Recircolation Tanks Drain*)
	SS2P_TNK_RingTankDrain : USINT := 13; (*Ring Tank Drain*)
	SS2P_TNK_PushBack : USINT := 14; (*PushBack In/Out*)
END_VAR
(*OPS Automatic Inlet Gate*)
VAR CONSTANT
	SS2P_OPS_InletGateManTest : USINT := 0; (*V4.A.A.1.6.12h*)
	SS2P_OPS_InletGateCommand : USINT := 1; (*V4.A.A.1.6.12h*)
END_VAR
(*v999hema*)
VAR CONSTANT
	SS2P_DOS_ModeCip : USINT := 0;
	SS2P_DOS_ModeDrain : USINT := 1;
	SS2P_DOS_ModeRinse : USINT := 2;
	SS2P_DOS_ModeProdFast : USINT := 3;
	SS2P_DOS_ModeQuickRinse : USINT := 4;
	SS2P_DOS_ModeFastRinse : USINT := 5;
	SS2P_DOS_SelLiftMan : USINT := 6;
	SS2P_DOS_ManualMMF205 : USINT := 7;
	SS2P_DOS_ManualMMF206 : USINT := 8;
	SS2P_DOS_ProbeAdjustment : USINT := 9;
	SS2P_DOS_CamDosByPass : USINT := 10;
	SS2P_DOS_CamDosInclusion : USINT := 11;
END_VAR
```

### SS3P_Constants.var - Selectors switch three positions constants
```iecst
(*SFT*)
VAR CONSTANT
	SS3P_SFT_FillingValveOpen : USINT := 0;
END_VAR
(*CAP*)
VAR CONSTANT
	SS3P_CAP_CapsRelease : USINT := 0;
	SS3P_CAP_UvLampChannelA : USINT := 1;
	SS3P_CAP_UvLampChannelB : USINT := 2;
	SS3P_CAP_UvLampChannelC : USINT := 3;
END_VAR
(*COP - Wash*)
VAR CONSTANT
	SS3P_COP_Shower : USINT := 0;
	SS3P_COP_NeckRinse : USINT := 1;
	SS3P_COP_ValveWash : USINT := 2;
	SS3P_COP_ColumnLubrification : USINT := 3;
	SS3P_COP_ValveWash2 : USINT := 4;
	SS3P_COP_HotWater : USINT := 5; (*//V4.A.A.1.7.4*)
END_VAR
(*CRW*)
VAR CONSTANT
	SS3P_CRW_CrownsRelease : USINT := 0;
	SS3P_CRW_Washing : USINT := 1;
	SS3P_CRW_ExtractorCleaning : USINT := 2;
END_VAR
(*v999hema*)
VAR CONSTANT
	SS3P_DOS_FillingValveOpen : USINT := 0;
END_VAR
```

### Package Logical/02_HMI - Human Machine Interface: interfaccia pannello operatore

### Program Logical/02_HMI/HMI (IEC) - HMI Main Program - C#6 - 200ms

#### HMI.sfc - Cyclic code
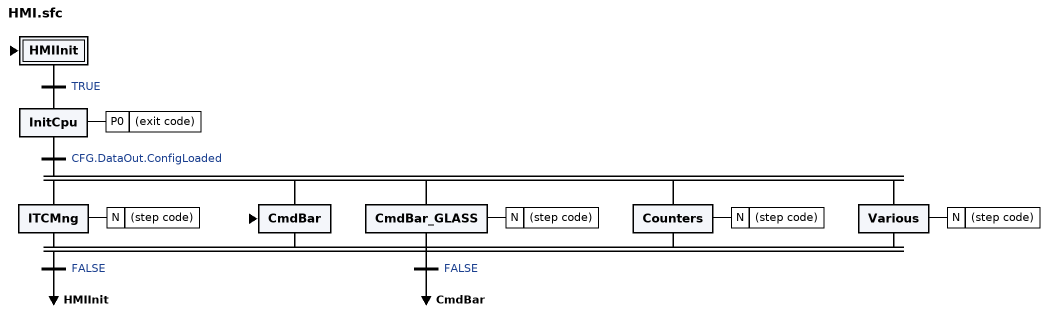
```iecst
PROGRAM _CYCLIC
INITIAL_STEP HMIInit:
END_STEP
TRANSITION FROM HMIInit TO InitCpu:=
TRUE
END_TRANSITION
STEP InitCpu:

END_STEP
EXIT_ACTION
HMI_MachinePlcVersion := 'V4.AA.200.8.0';

//V4.A.A.1.6.13
VAR_SafetyVersionTemp := UINT_TO_USINT(swapUINT(PI.SwVer1));
itoa(VAR_SafetyVersionTemp, ADR(VAR_SafetyVersionData1));

VAR_SafetyVersionTemp := UINT_TO_USINT(PI.SwVer1);
itoa(VAR_SafetyVersionTemp, ADR(VAR_SafetyVersionData2));

VAR_SafetyVersionTemp := UINT_TO_USINT(swapUINT(PI.SwVer2));
itoa(VAR_SafetyVersionTemp, ADR(VAR_SafetyVersionData3));

VAR_SafetyVersionTemp :=  UINT_TO_USINT(PI.SwVer2);
itoa(VAR_SafetyVersionTemp, ADR(VAR_SafetyVersionData4));

strcat(ADR(HMI_MachineSafetyVersion), ADR('V'));
strcat(ADR(HMI_MachineSafetyVersion), ADR(VAR_SafetyVersionData1));
strcat(ADR(HMI_MachineSafetyVersion), ADR('.'));
strcat(ADR(HMI_MachineSafetyVersion), ADR(VAR_SafetyVersionData2));
strcat(ADR(HMI_MachineSafetyVersion), ADR('.'));
strcat(ADR(HMI_MachineSafetyVersion), ADR(VAR_SafetyVersionData3));
strcat(ADR(HMI_MachineSafetyVersion), ADR('.'));
strcat(ADR(HMI_MachineSafetyVersion), ADR(VAR_SafetyVersionData4));
END_ACTION
TRANSITION FROM InitCpu TO (ITCMng,CmdBar,CmdBar_GLASS,Counters,Various):=
CFG.DataOut.ConfigLoaded
END_TRANSITION
STEP ITCMng:
(* ITC *)
HMI_ITCMng;
END_STEP
STEP CmdBar:
END_STEP
STEP CmdBar_GLASS:
// Command Bar - Fixed Visibility and Partner Visibility
HMI_CommandBar_Visibility_GLASS;
//
//	(* Command Bar - Command from HMI and Partner *)
HMI_CommandBar_Command_GLASS;
//
//	(* Command Bar - Enable from PLC and Partner *)
HMI_CommandBar_Enable_GLASS;
//
//	(* Command Bar - State from PLC and Partner *)
HMI_CommandBar_Status_GLASS;

END_STEP
TRANSITION FROM CmdBar_GLASS TO CmdBar:=
FALSE
END_TRANSITION
(* @SFCISJUMP := 'CmdBar' *)
STEP Counters:
(* Counter *)
HMI_CounterMng;
END_STEP
STEP Various:
HMI_SS2P[SS2P_HMI_DeviceEnable].Visibility	:= TRUE;
HMI_SS2P[SS2P_HMI_DeviceEnable].Enable		:= TRUE;
HMI_SS2P[SS2P_HMI_DeviceEnable].LampON		:= HMI_SS2P[SS2P_HMI_DeviceEnable].ON;

HMI_SS2P[SS2P_HMI_SelEnable].Visibility	:= TRUE;
HMI_SS2P[SS2P_HMI_SelEnable].Enable		:= TRUE;
HMI_SS2P[SS2P_HMI_SelEnable].LampON		:= HMI_SS2P[SS2P_HMI_SelEnable].ON;

(* HMI-PLC Communication WatchDog *)
TMR_TON_WatchDogOn(IN:= NOT HMI_WatchDog, PT := t#2s);

TMR_TON_WatchDogOff(IN:= HMI_WatchDog, PT := t#2s);

IF TMR_TON_WatchDogOn.Q THEN
	HMI_WatchDog := TRUE;
ELSIF TMR_TON_WatchDogOff.Q THEN
	HMI_WatchDog := FALSE;
END_IF
END_STEP
TRANSITION FROM (ITCMng,CmdBar,Counters,Various) TO HMIInit:=
FALSE
END_TRANSITION
(* @SFCISJUMP := 'HMIInit' *)
END_PROGRAM
```

#### Variables.var - Local variables
```iecst
VAR
	HMI_ITC_PageData : REFERENCE TO HMI_ITC_Data_Type;
	HMI_ITC_PartnerOld : USINT;
	VAR_CoupledModality : SR := (Q1:=TRUE);
	VAR_BlrCombiModality : SR;
	VAR_LbrCombiModality : SR;
	VAR_ActCombiModality : SR; (*V4.A.A.1.6.12*)
	VAR_ContUnblock1 : SR;
	VAR_ContUnblock2 : SR;
	VAR_ContBlock1 : SR;
	VAR_ContBlock2 : SR;
	TMR_TON_WatchDogOn : TON;
	TMR_TON_WatchDogOff : TON;
	VAR_Temp_HmiPartnerID : USINT;
	VAR_ITCindex : USINT;
	RCPType_APCO : REAL;
	VAR_CoTypeOfChangeCFG : INT;
	HMI_CounterPartialDataPageDB : REFERENCE TO ARRAY[0..15] OF Counters_Type;
	HMI_CounterPartialCfgPageDB : REFERENCE TO ARRAY[0..15] OF HmiCounterData_Type;
	HMI_CounterTotalDataPageDB : REFERENCE TO ARRAY[0..15] OF Counters_Type;
	HMI_CounterTotalCfgPageDB : REFERENCE TO ARRAY[0..15] OF HmiCounterData_Type;
	HMI_CounterPageCategory : USINT;
	HMI_WatchDog : BOOL;
	VAR_BlrCombiModalityReset : BOOL; (*V4.A.A.1.6.12h*)
	VAR_SafetyVersionTemp : USINT; (*V4.A.A.1.6.13*)
	VAR_SafetyVersionData1 : STRING[2] := '0'; (*V4.A.A.1.6.13*)
	VAR_SafetyVersionData2 : STRING[2] := '0'; (*V4.A.A.1.6.13*)
	VAR_SafetyVersionData3 : STRING[2] := '0'; (*V4.A.A.1.6.13*)
	VAR_SafetyVersionData4 : STRING[2] := '0'; (*V4.A.A.1.6.13*)
END_VAR
```

#### HMI_AID_Loading.st
```iecst
ACTION HMI_AID_Loading:
	HMI_CmdBar_PB;
	HMI_PB;
	HMI_SS2P;
	HMI_SS2P_Custom;//V4.A.A.1.6.13
END_ACTION
```

#### HMI_ALR_Loading.st
```iecst
ACTION HMI_ALR_Loading:
	HMI_ALR;
	HMI_MSG;
END_ACTION
```

#### HMI_RNS_Loading.st
```iecst
ACTION HMI_RNS_Loading:
	HMI_RNS_PB;
	HMI_RNS_SS2P;
	HMI_RNS_SS3P;
//	HMI_RNS_State;

	HMI_202DSB;

	HMI_205DSB;//V4.A.A.1.7.0

	HMI_206CPB;//V4.A.A.1.7.0
	HMI_296CPB;//V4.A.A.1.7.0
	HMI_297CPB;//V4.A.A.1.7.0
	HMI_298CPB;//V4.A.A.1.7.0
	HMI_299CPB;//V4.A.A.1.7.0

	HMI_296CPB_I;//V4.A.A.1.7.0
	HMI_297CPB_I;//V4.A.A.1.7.0

	HMI_RNS_NozzleData;//V4.A.A.1.7.0
	HMI_RNS_ManualSelection;//V4.A.A.1.7.0
	HMI_RNS_TypeCFG;//V4.A.A.1.7.0
	HMI_RNS_MultiChoiceMng;//V4.A.A.1.7.0
END_ACTION
```

#### HMI_CAP_Loading.st
```iecst
ACTION HMI_CAP_Loading:
	HMI_CAP_State;
	HMI_CAP_PB;
	HMI_CAP_SS2P;
	HMI_CAP_SS3P;
	HMI_CAP_CapsTypeCFG;
	HMI_CAP_ManualCapsSelection;
	HMI_CAP_ConfigStructure;
	HMI_CAP_GreasingState;
	HMI_CAP_GreasingState2;		//V4.A.A.1.6.11
	HMI_CAP_GreasingData;
	HMI_CAP_GreasingData2;		//V4.A.A.1.6.11
	HMI_CAP_BufferPresent;//V1.3
	HMI_CAP_MultiChoiceMng; //v1.4
	HMI_CAP_Brush; //v1.4
	HMI_CAP_DataCfg; //v1.4
	HMI_CAP_BufferAdjust; //V4.A.A.1.6.11
	HMI_CAP_HRM; //V4.A.A.1.6.11

	//MOTORS
	HMI_206MMR;
	HMI_206MMRBrake;
	HMI_207MMR;
	HMI_229MMR; //V4.A.A.1.6.11
	HMI_230MMR;
	HMI_231MMR; //V4.A.A.1.6.11
	HMI_212MMR;
	HMI_213MMR;
	HMI_214MMR;
	HMI_215MMR;
	HMI_202GPE;
	HMI_203GPE;	//V4.A.A.1.6.11

	//SIKO MOTOR(*V1.61*)
	HMI_CAP_SikoMotor;//V1.61
	HMI_CAP_SikoMotorSetPointEnable;//V1.61

	//IONIZER
	HMI_201DRC;

	//DRIVERS
	HMI_VFD_206MMR;
	HMI_VFD_207MMR;
	HMI_VFD_230MMR;
	HMI_VFD_212MMR;
	HMI_VFD_213MMR;
	HMI_VFD_214MMR;
	HMI_VFD_215MMR;

	//VALVES
	HMI_201CPC;
	HMI_202CPC;
	HMI_205CPC;
	HMI_206CPC;
	HMI_207CPC;
	HMI_212CPC;
	HMI_213CPC;
	HMI_214CPC;
	HMI_215CPC;
	HMI_216CPC;
	HMI_217CPC;
	HMI_218CPC;
	HMI_219CPC;
	HMI_220CPC;
	HMI_221CPC;
	HMI_222CPC;
	HMI_223CPC;
	HMI_224CPC;
	HMI_225CPC;
	HMI_226CPC;
	HMI_227CPC;
	HMI_228CPC;
	HMI_229CPC;
	HMI_232CPC;  //V. 1.1
	HMI_233CPC;  //V4.A.A.1.6.11
	HMI_235CPC; //v1.7.4
	HMI_236CPC; //v1.7.4
	HMI_237CPC; //v1.7.4
	HMI_238CPC; //v1.7.4
	HMI_201EVC;
	HMI_203EVC;
	HMI_207EVC;
	HMI_209EVC;
	HMI_210EVC;
	HMI_211EVC;
	HMI_212EVC;
	HMI_213EVC;
	HMI_214EVC;
	HMI_215EVC;
	HMI_216EVC;
	HMI_227EVC; //v1.7.4
	HMI_228EVC; //1.7.4
	HMI_229EVC; //v1.7.4
	HMI_203EVF;

	//SENSOR
	HMI_202DSC;
	HMI_204DSC;
	HMI_205DSC;
	HMI_210DSC;  //V4.A.A.1.7.1
	HMI_211DSC;  //V4.A.A.1.7.1
	HMI_216DSC;
	HMI_217DSC;
	HMI_218DSC;
	HMI_219DSC;
	HMI_220DSC;
	HMI_221DSC;
	HMI_222DSC;
	HMI_223DSC;
	HMI_224DSC;
	HMI_225DSC;
	HMI_226DSC;
	HMI_227DSC;
	HMI_228DSC;
	HMI_229DSC;
	HMI_230DSC;
	HMI_231DSC;
	HMI_232DSC;
	HMI_233DSC;
	HMI_234DSC;
	HMI_235DSC;
	HMI_236DSC;
	HMI_237DSC;
	HMI_238DSC;
	HMI_239DSC;
	HMI_240DSC;
	HMI_241DSC;
	HMI_242DSC;
	HMI_243DSC;
	HMI_244DSC;
	HMI_245DSC;
	HMI_246DSC;
	HMI_247DSC;
	HMI_248DSC;
	HMI_249DSC;
	HMI_250DSC;
	HMI_251DSC;
	HMI_252DSC;
	HMI_253DSC;
	HMI_254DSC;
	HMI_255DSC;
	HMI_256DSC;
	HMI_257DSC;
	HMI_258DSC;	//V4.A.A.1.6.11
	HMI_259DSC;	//V4.A.A.1.6.11
	HMI_260DSC;	//V4.A.A.1.6.11
	HMI_261DSC; //V4.A.A.1.6.11
	HMI_262DSC; //V4.A.A.1.6.11
	HMI_263DSC; //V4.A.A.1.6.11
	HMI_264DSC;//V4.A.A.1.6.12h
	HMI_266DSC; //v1.7.4
	HMI_267DSC; //v1.7.5
	HMI_268DSC; //v1.7.5
	HMI_270DSC; //v1.7.4
	HMI_ST3A;//(*//V4.A.A.1.6.12*)
	HMI_ST3B;//(*//V4.A.A.1.6.12*)

END_ACTION
```

#### HMI_CRW_Loading.st
```iecst
ACTION HMI_CRW_Loading:
	HMI_CRW_PB;
	HMI_CRW_SS2P;
	HMI_CRW_SS3P;
	HMI_CRW_CrownsTypeCFG;

	//VALVES
	HMI_230CPC;
	HMI_231CPC;
	HMI_231EVC;(*master nuovo*)
	HMI_205EVC;

	//SENSORS
	HMI_253DSC;
	HMI_254DSC;
	HMI_255DSC;
	HMI_256DSC;
	HMI_274DSC;(*master nuovo*)

END_ACTION
```

#### HMI_CO_Loading.st
```iecst
ACTION HMI_CO_Loading:
	HMI_APCO;
	HMI_APCO_TypeOfChangeCFG;
	HMI_CO_SS2P;
	HMI_APCO_TypeOfChange;
END_ACTION
```

#### HMI_COP_Loading.st
```iecst
ACTION HMI_COP_Loading:
	HMI_COP_StatusWidget;
	HMI_COP_PB;
	HMI_COP_SS2P;
	HMI_COP_SS3P;
	HMI_COP_Rcp;
	HMI_COP_RcpTemp;
	HMI_COP_RcpSelection;
	HMI_COP_RcpInfo;
	HMI_COP_State;
	HMI_COP_ZoneCfg;
	HMI_RCP_COP_Mngt;
	HMI_COP_PhaseTypeCFG;
	HMI_COP_FuTypeCFG;
	HMI_COP_FuGunTypeCFG;
	HMI_COP_FuDrainableCFG;
	HMI_COP_ITC;
	HMI_COP_OptPlangerPresent;//VRMA
	HMI_RCP_COP_SelectedRecipeName; //v999hema
END_ACTION
```

#### HMI_CSR_Loading.st
```iecst
ACTION HMI_CSR_Loading:
	HMI_CSR_PB;
	HMI_CSR_SS2P;
	HMI_CSR_SS3P;
	HMI_LTK;
	HMI_CSR_State;
	HMI_CSR_SCU;
	HMI_CSR_Column;
	HMI_CSR_TnkLinftingMotor;
	HMI_CSR_Data;
	HMI_2808M1;(*master nuovo*)
	HMI_204CPC;(*master nuovo*)
	HMI_2809M2;(*master nuovo*)
	HMI_YV26;(*master nuovo*)
	HMI_YV39;(*master nuovo*)
	HMI_SQ26;(*master nuovo*)
	HMI_SQ45A2;(*master nuovo*)
	HMI_SQ45A1;(*master nuovo*)
	HMI_SQ70;(*master nuovo*)
	HMI_SQ5;(*master nuovo*)
	HMI_SQ6;(*master nuovo*)
	HMI_CSR_SikoActualPosition;//V1.61
	HMI_CSR_SikoConveyorData;//V1.61
	HMI_CSR_SikoGuideData;//V1.61

END_ACTION
```

#### HMI_DMC_Loading.st
```iecst
ACTION HMI_DMC_Loading:
	HMI_DMC_SS2P;
	HMI_DMC_PB;//v999
	HMI_DMC_StepActual; // NOT USED
	HMI_DMC_State;
	HMI_DMC_Number;
	HMI_DMC_InsertionSensor;
	HMI_DMC_InsertionPiston;
	HMI_DMC_Installed;
	HMI_DMC_Visualization;
	HMI_205RVF;
	HMI_DMC_OkFromOperatorCheck;
	HMI_DMC_AbortFromOperatorCheck;
	HMI_DMC_ManModeStatus;//v999
	HMI_DMC_AutoModeStatus;
	HMI_DMC_TankHeightPosOk;//
	HMI_DMC_Sector1LastValveNum;//v999
	HMI_DMC_Sector2FirstValveNum;//v999
	HMI_DMC_Sector2LastValveNum;//v999
END_ACTION
```

#### HMI_GNS_Loading.st
```iecst
ACTION HMI_GNS_Loading:
	HMI_204PSF;
	HMI_201PTF;
	HMI_204PTF;
	HMI_205PTF;
	HMI_206PTF;
	HMI_Beacon;
	HMI_BeaconHome; //V4.A.A.1.6.8
	HMI_GNS_LadderRestPosition;
	HMI_202QTB;//v1.7.4
	HMI_202QTE;//v1.7.4
	HMI_201QTB;//v1.7.4
	HMI_201QTE;//v1.7.4
END_ACTION
```

#### HMI_ICO_Loading.st
```iecst
ACTION HMI_ICO_Loading:
	HMI_ICO;
END_ACTION
```

#### HMI_ITC_Loading.st
```iecst
ACTION HMI_ITC_Loading:
	HMI_ITC_Page;
	HMI_ITC_PageData ACCESS (ADR(HMI_ITC_PageDB[11]));
	HMI_ITC_Partner_CFG;
END_ACTION
```

#### HMI_MAU_Loading.st
```iecst
ACTION HMI_MAU_Loading:
	HMI_MAU_PB;
	HMI_MAU_SS2P;(*master nuovo*)
	HMI_GrLb_Loading;
	HMI_WhRoom_Loading;
	HMI_MAU_Safety_Loading;
	HMI_LbCon_Loading;(*master nuovo*)
	HMI_LftCon_Loading;
	HMI_UPS_Loading;
	HMI_MAU_Plc;
	HMI_Exhauster_Loading; //v1.7.4
END_ACTION

ACTION HMI_GrLb_Loading:
	HMI_201GPE;
	HMI_GrLb_PB;
	HMI_GrLb_Data;
	HMI_GrLb_Data2;		//V4.A.A.1.6.11
END_ACTION

ACTION HMI_LbCon_Loading:(*master nuovo*)
	HMI_LbCon_PB;(*master nuovo*)
	HMI_MAU_ChlRns;(*master nuovo*)
END_ACTION
ACTION HMI_Tray_Loading:
	//v1.4
	HMI_227CPB;
	HMI_209DSF;
END_ACTION

ACTION HMI_LftCon_Loading:
	HMI_LftCon_SS2P;
	HMI_203RVF;
END_ACTION

ACTION HMI_WhRoom_Loading:
	HMI_WhRoom_SS2P;
	HMI_FanBase;
	HMI_FanFiller;
	HMI_FanRinser;
	HMI_FanTransfer;
	HMI_204PTE;
	HMI_205PTE;
	HMI_206PTE;
	HMI_207PTE;//1.7.6
END_ACTION

ACTION HMI_UPS_Loading:
	HMI_UPS_ShutdownRequest;
END_ACTION

ACTION HMI_MAU_Safety_Loading:
	HMI_SL_Info;
	HMI_SL_PB;
END_ACTION

ACTION HMI_MAU_Plc:
	HMI_TimeZoneOffset;
	HMI_SDM_RequestInit;//1.7.2b
 	HMI_SDM_PLCAvailable;//1.7.2b
	HMI_SDM_MachineStopped;//1.7.2b
END_ACTION

ACTION HMI_Exhauster_Loading: //v1.7.4
HMI_AFE;
HMI_VFD_AFE;
END_ACTION
```

#### HMI_MNM_Loading.st
```iecst
ACTION HMI_MNM_Loading:
	HMI_MNM_PB;
	HMI_MNM_MachineSpeedAct;
	HMI_MNM_MachineSpeedReq;
	HMI_MNM_MinMachineSpeed;
	HMI_MNM_MinMachineJogSpeed := CST_JogMinimumSpeed;
	HMI_MNM_MaxMachineJogSpeed := CST_JogMaximumSpeed;
	HMI_MNM_MinInMotionAdjustement;
	HMI_MNM_MaxInMotionAdjustement;
	HMI_MNM_MaxMachineSpeed;
	HMI_MNM_AxisPositionOffset;
	HMI_MNM_AxisStepByStepOffset;
	HMI_MNM_AxisInMotionAdjustment;
	HMI_MNM_MachinePitch;
	HMI_MNM_AxisSelected;
	HMI_MNM_ConveyorSpeed;
	HMI_MNM_MachinePosition;
	HMI_MNM_FlrSpeedWidget;
	HMI_MNM_SmrSpeedWidget;
	HMI_MNM_MachineRunning;

	HMI_ContainerFallInlet1;
	HMI_ContainerFallInlet2;
	HMI_NoContainerInlet1;
	HMI_NoContainerInlet2;
	HMI_OutletFull;
	//MOTORS
	HMI_OutCvr;
	HMI_InCvr;(*master nuovo*)
	//DRIVERS
	HMI_VFD_OutCvr;
	HMI_VFD_InCvr;(*master nuovo*)
	//SENSORS
	HMI_236DSE;
	HMI_230DSE;
	HMI_241DSE;

	//V4.A.A.1.7.0
	HMI_MNM_CamName;

	HMI_MNM_NumOfDmcInTangentSector1;
	HMI_MNM_NumOfDmcInTangentSector2;
END_ACTION
```

#### HMI_MNT_Loading.st
```iecst
ACTION HMI_MNT_Loading:
	HMI_MNT;
END_ACTION
```

#### HMI_OPS_Loading.st
```iecst
ACTION HMI_OPS_Loading:
	HMI_OPS_Zone;
	HMI_OPS_Door;
	HMI_OPS_DoorCabinet;//V1.3
	HMI_OPS_DoorCabinet_Visibility;//V4.A.A.1.7.0
	HMI_OPS_Euchner;//V1.3
	HMI_OPS_SafetySwitch;//V4.A.A.1.7.1
	HMI_OPS_Emergency;
	HMI_OPS_EmergencyBlower;
	HMI_OPS_EmergencyLabeller;
	HMI_OPS_EmergencyConveyor;
	HMI_OPS_EmergencyNitrodoser;
	HMI_OPS_EmergencyCapsFeeder;
	HMI_OPS_EmergencyCrownFeeder;
	HMI_OPS_Jog;
	HMI_OPS_JogFwExt;//vrma106
	HMI_OPS_ModeSelectorAdjustment;
	HMI_OPS_ModeSelectorJog; //V4.A.A.1.6.13
	HMI_OPS_ModeSelectorAuto; //V4.A.A.1.6.13
	HMI_OPS_GateDoor;
	HMI_OPS_SafetyWidget;
	HMI_OPS_Pictogram;
	HMI_OPS_PB;
	HMI_OPS_SS2P;//V4.A.A.1.6.12h
	HMI_OPS_ZoneComboString;
	HMI_OPS_Cfg;
	HMI_OPS_BufferDoor;
	HMI_OPS_BufferZone;
	HMI_207EVF;//V4.A.A.1.6.12
	HMI_209EVF;
	HMI_208CPF;//V4.A.A.1.6.12
	HMI_208DSFX;//V4.A.A.1.6.12
	HMI_208DSFY;//V4.A.A.1.6.12
	HMI_209DSFX;//V4.A.A.1.6.12
	HMI_209DSFY;//V4.A.A.1.6.12
END_ACTION
```

#### HMI_OPT_Loading.st
```iecst
ACTION HMI_OPT_Loading:
	HMI_OPT_SS2P;
END_ACTION
```

#### HMI_PAO_Loading.st
```iecst
ACTION HMI_PAO_Loading:
	HMI_PAO;
	HMI_CFG_Display;
	HMI_CFG_Reset;
	HMI_CFG_Selection;
END_ACTION
```

#### HMI_SFT_Loading.st
```iecst
ACTION HMI_SFT_Loading:
	HMI_SFT_PB;
	HMI_SFT_SS2P;
	HMI_SFT_SS3P;

	//VALVES
	HMI_207CPB; //V4.A.A.1.6.11

	//COUNTERS
	HMI_StepAcquisition;
	HMI_CounterPartialCfgPageDB		ACCESS	(ADR(HMI_CounterCfgPartial.MachineCounters));
	HMI_CounterPartialDataPageDB	ACCESS	(ADR(HMI_CounterDataPartial.MachineCounters));
	HMI_CounterTotalCfgPageDB		ACCESS	(ADR(HMI_CounterCfgTotal.MachineCounters));
	HMI_CounterTotalDataPageDB		ACCESS	(ADR(HMI_CounterDataTotal.MachineCounters));
	HMI_TotalBottleProduced;

	//PHOTOCELLS
	HMI_201DSC;
	HMI_202DSF;
	HMI_203DSF;
	HMI_204DSF;
	HMI_207DSF;
	HMI_208DSF;
	HMI_204DSB; //v999hema
	HMI_205DSB; //v999hema
	HMI_201CPB;
	//Auto DMC
	HMI_ProductionSensorCheck1;
	HMI_ProductionSensorCheck2;
	HMI_ProductionSensorCheck3;

	//Bottle Burst
	HMI_SFT_BurstData;

	HMI_298DSB;//V4.A.A.1.7.0
	HMI_299DSB;//V4.A.A.1.7.0

	HMI_SFT_NumberOfDummyInError;
	HMI_SFT_NumberOfDmcInPosCheck;
END_ACTION
```

#### HMI_TNK_Loading.st
```iecst
ACTION HMI_TNK_Loading:
	HMI_FMC_ActualFlowRate;
END_ACTION
```

#### HMI_Device_Loading.st
```iecst
ACTION HMI_Valves_Loading:
	HMI_AVB;
	HMI_EVB; //v1.7.4
	HMI_HVB;//V4.A.A.1.6.12
	HMI_RVB;
	HMI_RMB;
	HMI_PID_RVB;
	HMI_PID_RMB;

	HMI_AVC;//V1.7.2
	HMI_HVC;//V1.7.2
	HMI_RVC;//V1.7.2
	HMI_RMC;//V1.7.2
	HMI_PID_RVC;//V1.7.2
	HMI_PID_RMC;//V1.7.2

	HMI_AVS;

	HMI_AVE;
	HMI_HVE;//V4.A.A.1.6.12
	HMI_RVE;
	HMI_RME;
	HMI_EHE;
	HMI_PID_RVE;
	HMI_PID_RME;

	HMI_AVX;
	HMI_RVX;
	HMI_RMX;
	HMI_PID_RVX;
	HMI_PID_RMX;

	HMI_AVJ;   	 //v999hema
	HMI_RVJ;
	HMI_PID_RVJ;
END_ACTION

ACTION HMI_Instruments_Loading:
	HMI_FSF;
	HMI_PSB;
	HMI_LSB;
	HMI_HSB;//V4.A.A.1.6.12
	HMI_FSB;
	HMI_CTB;
	HMI_QTB;
	HMI_FTB;
	HMI_TTB;
	HMI_PTB;
	HMI_LTB;
	HMI_PID_RVB;
	HMI_PID_RMB;

	HMI_PSC;//V1.7.2
	HMI_LSC;//V1.7.2
	HMI_HSC;//V1.7.2
	HMI_FSC;//V1.7.2
	HMI_CTC;//V1.7.2
	HMI_QTC;//V1.7.2
	HMI_FTC;//V1.7.2
	HMI_TTC;//V1.7.2
	HMI_PTC;//V1.7.2
	HMI_LTC;//V1.7.2
	HMI_PID_RVC;//V1.7.2
	HMI_PID_RMC;//V1.7.2

	HMI_PSE;
	HMI_LSE;
	HMI_FSE;
	HMI_CTE;
	HMI_QTE;
	HMI_FTE;
	HMI_TTE;
	HMI_PTE;
	HMI_LTE;
	HMI_HSE;//V4.A.A.1.6.12
	HMI_PID_RVE;
	HMI_PID_RME;

	HMI_PSX;
	HMI_LSX;
	HMI_FSX;
	HMI_CTX;
	HMI_QTX;
	HMI_FTX;
	HMI_FTE; //v1.1
	HMI_TTX;
	HMI_PTX;
	HMI_LTX;
	HMI_PID_RVX;
	HMI_PID_RMX;

	HMI_QSB; //v1.7.4

	//v999hema
	HMI_LSJ200L;
	HMI_LSJ200M;
	HMI_LSJ200H;
	HMI_LSJ201H;
	HMI_LSJ202H;
	HMI_FSJ;
	HMI_TTJ;
	HMI_LTJ;

	HMI_205MEF;
	HMI_206MEF;
	HMI_215DSF;
	HMI_216DSF;
	HMI_217DSF;
	HMI_210DSX;
	HMI_211DSX;
	HMI_212DSF;
	HMI_213DSF;

	HMI_224DSB; //v999hema
	HMI_225DSB;
	HMI_226DSB;
	HMI_227DSB;

	HMI_210CPF;
	HMI_211CPF;
	HMI_210PTF;

END_ACTION

ACTION HMI_Pumps_Loading:
	HMI_MMB;
	HMI_VFD_MMB;
	HMI_PPB;
	HMI_PID_PPB;
	HMI_VFD_PPB;

	HMI_MMC;//v1.7.2
	HMI_VFD_MMC;//v1.7.2
	HMI_PPC;//v1.7.2
	HMI_PID_PPC;//v1.7.2
	HMI_VFD_PPC;//v1.7.2

	HMI_MME;
	HMI_VFD_MME;
	HMI_PPE;
	HMI_PID_PPE;
	HMI_VFD_PPE;

	HMI_MMX;
	HMI_VFD_MMX;
	HMI_PPX;
	HMI_PID_PPX;
	HMI_VFD_PPX;

	HMI_206PPB;//v1.7.4
	HMI_206PPB_Dos;//v1.7.4
	HMI_MMF; //v999hema
	HMI_MMJ;
	HMI_VFD_MMF;
	HMI_VFD_MMJ;
	HMI_PPJ;
	HMI_VFD_PPJ;
	HMI_PPJ203;
	HMI_PID_PPJ;
END_ACTION
```

#### HMI_Variables_Loading.st
```iecst
ACTION HMI_Variables_Loading:
	HMI_MachineId;
	HMI_MachinePlcVersion; //V4.A.A.1.6.13
	HMI_MachineSafetyVersion; //V4.A.A.1.6.13
	HMI_ScreenTouched;
	HMI_ApcoPresent;
	HMI_IcoPresent;
	HMI_CounterHome; //V4.A.A.1.6.8
END_ACTION
```

#### HMI_BTC_Loading.st - not listed in the package file held
```iecst
ACTION HMI_BTC_Loading:
	HMI_BTC_PB;
	HMI_BTC_SS2P;
	HMI_BTC_SS3P;
	HMI_BTC_State;
	HMI_BTC_UVL;
END_ACTION
```

#### Package Logical/02_HMI/HMI/HMI_CmdBar - HMI Command Bar Configuration

#### Command_Bar_GLASS.st
```iecst
ACTION HMI_CommandBar_Visibility_GLASS:
	HMI_CmdBar_PB[PB_MixerProcessStart].Visibility		:= CFG_Par.Process.BlendFill;
	HMI_CmdBar_PB[PB_FillerProcessStart].Visibility		:= NOT CFG_Par.Process.BlendFill;(*master nuovo*)
	HMI_CmdBar_PB[PB_FillerDoorUnlock].Visibility		:= TRUE;
	HMI_CmdBar_PB[PB_ContainerBlock1].Visibility		:= TRUE;
	HMI_CmdBar_PB[PB_ContainerRelease1].Visibility		:= TRUE;

END_ACTION

ACTION HMI_CommandBar_Command_GLASS:
	HMI_CmdBar_PB[PB_MixerProcessStart].Command			:= HMI_CmdBar_PB[PB_MixerProcessStart].ON;// v4 200.2.0 eliminate logiche combi
	HMI_CmdBar_PB[PB_FillerProcessStart].Command		:= HMI_CmdBar_PB[PB_FillerProcessStart].ON;// v4 200.2.0 eliminate logiche combi
	HMI_CmdBar_PB[PB_FillerDoorUnlock].Command			:= HMI_CmdBar_PB[PB_FillerDoorUnlock].ON;// v4 200.2.0 eliminate logiche combi

	VAR_ContUnblock1(
	SET1	:= EDGEPOS(HMI_CmdBar_PB[PB_ContainerRelease1].ON) AND NOT VAR_ContUnblock1.Q1,
	RESET	:= (EDGEPOS(HMI_CmdBar_PB[PB_ContainerRelease1].ON OR SFT.DataOut.ManualContainersReleaseEnable) AND VAR_ContUnblock1.Q1) OR EDGEPOS(HMI_CmdBar_PB[PB_ContainerBlock1].ON) OR EDGEPOS(SFT.DataOut.COPInletContConvEmptyRunning)(*master nuovo*)

	);

	VAR_ContBlock1(
	SET1	:= EDGEPOS(HMI_CmdBar_PB[PB_ContainerBlock1].ON) AND NOT VAR_ContBlock1.Q1,
	RESET	:= (EDGEPOS(HMI_CmdBar_PB[PB_ContainerBlock1].ON) AND VAR_ContBlock1.Q1) OR EDGEPOS(HMI_CmdBar_PB[PB_ContainerRelease1].ON)
	);

	HMI_CmdBar_PB[PB_ContainerBlock1].Command			:= VAR_ContBlock1.Q1;
	HMI_CmdBar_PB[PB_ContainerRelease1].Command			:= VAR_ContUnblock1.Q1;
	HMI_CmdBar_PB[PB_MixerProcessStart].Command			:= HMI_CmdBar_PB[PB_MixerProcessStart].ON;// v4 200.2.0 eliminate logiche combi

END_ACTION

ACTION HMI_CommandBar_Enable_GLASS:
	HMI_CmdBar_PB[PB_MixerProcessStart].Enable			:= SEL(CFG_Par.Process.BlendFill,SkdFlr.HMI_ProcessStartEnable,CrbFlr.HMI_ProcessStartEnable);;(*master nuovo*)
	HMI_CmdBar_PB[PB_FillerProcessStart].Enable			:= SEL(CFG_Par.Process.BlendFill,SkdFlr.HMI_ProcessStartEnable,CrbFlr.HMI_ProcessStartEnable);
	HMI_CmdBar_PB[PB_FillerDoorUnlock].Enable			:= NOT PO.ReleaseEnable;//vrma
	HMI_CmdBar_PB[PB_ContainerBlock1].Enable			:= TRUE;
	HMI_CmdBar_PB[PB_ContainerRelease1].Enable			:= TRUE; // leo(SFT.DataOut.ManualContainersReleaseEnable OR HMI_CmdBar_PB[PB_ContainerRelease1].Command) AND NOT SFT.DataOut.COPInletContConvEmptyRunning;

END_ACTION

ACTION HMI_CommandBar_Status_GLASS:
	HMI_CmdBar_PB[PB_MixerProcessStart].LampON			:= SEL(CFG_Par.Process.BlendFill,SkdFlr.HMI_ProcessStartLampOn, CrbFlr.HMI_ProcessStartLampOn);	(*master nuovo*)
	HMI_CmdBar_PB[PB_FillerProcessStart].LampON			:= SEL(CFG_Par.Process.BlendFill, SkdFlr.HMI_ProcessStartLampOn, CrbFlr.HMI_ProcessStartLampOn);
	HMI_CmdBar_PB[PB_FillerDoorUnlock].LampON			:= OPS.DataOut.HMIDoorUnlock;
	HMI_CmdBar_PB[PB_FillerProcessStart].Blink			:= SEL(CFG_Par.Process.BlendFill, SkdFlr.HMI_ProcessStartBlink, CrbFlr.HMI_ProcessStartBlink);
	HMI_CmdBar_PB[PB_ContainerBlock1].Blink				:= VAR_ContBlock1.Q1 AND NOT HMI_CmdBar_PB[PB_ContainerBlock1].Command;
	HMI_CmdBar_PB[PB_ContainerRelease1].LampON			:= HMI_CmdBar_PB[PB_ContainerRelease1].Command;
	HMI_CmdBar_PB[PB_ContainerBlock1].LampON			:= HMI_CmdBar_PB[PB_ContainerBlock1].Command;

END_ACTION
```

#### Command_Bar_CAN.st
```iecst
ACTION HMI_CommandBar_Visibility_CAN:
	HMI_CmdBar_PB[PB_FillerSeamerCoupled].Visibility	:= TRUE;
	HMI_CmdBar_PB[PB_FillerStartStop].Visibility		:= TRUE;
	HMI_CmdBar_PB[PB_SeamerStartStop].Visibility		:= TRUE;
	HMI_CmdBar_PB[PB_FillerProcessStart].Visibility		:= TRUE;
	HMI_CmdBar_PB[PB_MixerProcessStart].Visibility		:= FALSE;
	HMI_CmdBar_PB[PB_ContainerBlock1].Visibility		:= TRUE;
	HMI_CmdBar_PB[PB_ContainerRelease1].Visibility		:= TRUE;
	HMI_CmdBar_PB[PB_ContainerBlock2].Visibility		:= CFG_Par.Motors.DoubleInlet;
	HMI_CmdBar_PB[PB_ContainerRelease2].Visibility		:= CFG_Par.Motors.DoubleInlet;
	HMI_CmdBar_PB[PB_FillerDoorUnlock].Visibility		:= TRUE;
	HMI_CmdBar_PB[PB_SeamerDoorUnlock].Visibility		:= TRUE;
END_ACTION

ACTION HMI_CommandBar_Command_CAN:
	VAR_CoupledModality(
	SET1	:= EDGEPOS(HMI_CmdBar_PB[PB_FillerSeamerCoupled].ON) AND NOT VAR_CoupledModality.Q1,
	RESET	:= EDGEPOS(HMI_CmdBar_PB[PB_FillerSeamerCoupled].ON) AND VAR_CoupledModality.Q1
	);

	VAR_ContUnblock1(
	SET1	:= EDGEPOS(HMI_CmdBar_PB[PB_ContainerRelease1].ON) AND NOT VAR_ContUnblock1.Q1,
	RESET	:= (EDGEPOS(HMI_CmdBar_PB[PB_ContainerRelease1].ON) AND VAR_ContUnblock1.Q1) OR EDGEPOS(HMI_CmdBar_PB[PB_ContainerBlock1].ON) OR EDGEPOS(SFT.DataOut.COPInletContConvEmptyRunning)
	);

	VAR_ContBlock1(
	SET1	:= EDGEPOS(HMI_CmdBar_PB[PB_ContainerBlock1].ON) AND NOT VAR_ContBlock1.Q1,
	RESET	:= (EDGEPOS(HMI_CmdBar_PB[PB_ContainerBlock1].ON) AND VAR_ContBlock1.Q1) OR EDGEPOS(HMI_CmdBar_PB[PB_ContainerRelease1].ON)
	);

	VAR_ContUnblock2(
	SET1	:= EDGEPOS(HMI_CmdBar_PB[PB_ContainerRelease2].ON) AND NOT VAR_ContUnblock2.Q1,
	RESET	:= (EDGEPOS(HMI_CmdBar_PB[PB_ContainerRelease2].ON) AND VAR_ContUnblock2.Q1) OR EDGEPOS(HMI_CmdBar_PB[PB_ContainerBlock2].ON) OR EDGEPOS(SFT.DataOut.COPInletContConvEmptyRunning)
	);

	VAR_ContBlock2(
	SET1	:= EDGEPOS(HMI_CmdBar_PB[PB_ContainerBlock2].ON) AND NOT VAR_ContBlock2.Q1,
	RESET	:= (EDGEPOS(HMI_CmdBar_PB[PB_ContainerBlock2].ON) AND VAR_ContBlock2.Q1) OR EDGEPOS(HMI_CmdBar_PB[PB_ContainerRelease2].ON)
	);

	HMI_CmdBar_PB[PB_FillerSeamerCoupled].Command	:= VAR_CoupledModality.Q1;
	HMI_CmdBar_PB[PB_FillerStartStop].Command		:= HMI_CmdBar_PB[PB_FillerStartStop].ON;
	HMI_CmdBar_PB[PB_SeamerStartStop].Command		:= HMI_CmdBar_PB[PB_SeamerStartStop].ON;
	HMI_CmdBar_PB[PB_FillerProcessStart].Command	:= HMI_CmdBar_PB[PB_FillerProcessStart].ON;
	HMI_CmdBar_PB[PB_MixerProcessStart].Command		:= HMI_CmdBar_PB[PB_MixerProcessStart].ON;
	HMI_CmdBar_PB[PB_ContainerBlock1].Command		:= VAR_ContBlock1.Q1 AND NOT (SFT.DataOut.COPInletContConvEmptyRunning XOR SFT.DataOut.COPInletContConvEmptyDone);
	HMI_CmdBar_PB[PB_ContainerRelease1].Command		:= VAR_ContUnblock1.Q1;
	HMI_CmdBar_PB[PB_ContainerBlock2].Command		:= VAR_ContBlock2.Q1 AND NOT (SFT.DataOut.COPInletContConvEmptyRunning XOR SFT.DataOut.COPInletContConvEmptyDone);
	HMI_CmdBar_PB[PB_ContainerRelease2].Command		:= VAR_ContUnblock2.Q1;
	HMI_CmdBar_PB[PB_FillerDoorUnlock].Command		:= HMI_CmdBar_PB[PB_FillerDoorUnlock].ON;
	HMI_CmdBar_PB[PB_SeamerDoorUnlock].Command		:= HMI_CmdBar_PB[PB_SeamerDoorUnlock].ON;
END_ACTION

ACTION HMI_CommandBar_Enable_CAN:
	IF MC_InputOutput.Network.Machine.Status.MultiModalityActive THEN
		HMI_CmdBar_PB[PB_FillerSeamerCoupled].Enable	:= NOT MC_InputOutput.Network.Filler.Status.ModuleRunning AND  NOT MC_InputOutput.Network.Outlet.Status.ModuleRunning;
	ELSE
		HMI_CmdBar_PB[PB_FillerSeamerCoupled].Enable	:= NOT MC_InputOutput.Network.Machine.Status.MachineRunning;
	END_IF

	HMI_CmdBar_PB[PB_FillerStartStop].Enable		:= OPS.DataOut.FlrModeSelectorAuto AND
														(MC_InputOutput.Network.Machine.Status.MultiModalityActive) AND NOT FmcFlr.FillingManualTestActive;
	//HMI_CmdBar_PB[PB_SeamerStartStop].Enable		:= OPS.DataOut.SmrModeSelectorAuto AND
	//													(MC_InputOutput.Network.Machine.Status.MultiModalityActive);
	//HMI_CmdBar_PB[PB_FillerProcessStart].Enable		:= SkdFlr.HMI_ProcessStartEnable AND HMI_CmdBar_PB[PB_FillerSeamerCoupled].Command AND NOT SMR.DataOut.CleaningReq;
	HMI_CmdBar_PB[PB_MixerProcessStart].Enable		:= FALSE;
	HMI_CmdBar_PB[PB_ContainerBlock1].Enable		:= TRUE;
	HMI_CmdBar_PB[PB_ContainerRelease1].Enable		:= (SFT.DataOut.ManualContainersReleaseEnable OR HMI_CmdBar_PB[PB_ContainerRelease1].Command) AND NOT SFT.DataOut.COPInletContConvEmptyRunning;
	HMI_CmdBar_PB[PB_ContainerBlock2].Enable		:= TRUE;
	HMI_CmdBar_PB[PB_ContainerRelease2].Enable		:= (SFT.DataOut.ManualContainersReleaseEnable OR HMI_CmdBar_PB[PB_ContainerRelease2].Command) AND NOT SFT.DataOut.COPInletContConvEmptyRunning;
	HMI_CmdBar_PB[PB_FillerDoorUnlock].Enable		:= NOT MC_InputOutput.Network.Machine.Status.MachineRunning AND NOT MC_InputOutput.Network.Filler.Status.ModuleRunning AND NOT TNK.DataOut.CipMode;
	HMI_CmdBar_PB[PB_SeamerDoorUnlock].Enable		:= NOT MC_InputOutput.Network.Machine.Status.MachineRunning AND NOT MC_InputOutput.Network.Outlet.Status.ModuleRunning;
END_ACTION

ACTION HMI_CommandBar_Status_CAN:
	HMI_CmdBar_PB[PB_FillerSeamerCoupled].LampON	:= HMI_CmdBar_PB[PB_FillerSeamerCoupled].Command;
	//HMI_CmdBar_PB[PB_FillerStartStop].LampON		:= MNM.DataOut.StartFlrLightFixRequest;
	//HMI_CmdBar_PB[PB_FillerStartStop].Blink			:= MNM.DataOut.StartFlrLightBlinkRequest;
	//HMI_CmdBar_PB[PB_SeamerStartStop].LampON		:= MNM.DataOut.StartSmrLightFixRequest;
	//HMI_CmdBar_PB[PB_SeamerStartStop].Blink			:= MNM.DataOut.StartSmrLightBlinkRequest;
	HMI_CmdBar_PB[PB_FillerProcessStart].LampON		:= SkdFlr.HMI_ProcessStartLampOn;
	HMI_CmdBar_PB[PB_FillerProcessStart].Blink		:= SkdFlr.HMI_ProcessStartBlink;
	HMI_CmdBar_PB[PB_MixerProcessStart].LampON		:= HMI_CmdBar_PB[PB_MixerProcessStart].Command;
	HMI_CmdBar_PB[PB_ContainerBlock1].LampON		:= HMI_CmdBar_PB[PB_ContainerBlock1].Command;
	HMI_CmdBar_PB[PB_ContainerBlock1].Blink			:= VAR_ContBlock1.Q1 AND NOT HMI_CmdBar_PB[PB_ContainerBlock1].Command;
	HMI_CmdBar_PB[PB_ContainerRelease1].LampON		:= HMI_CmdBar_PB[PB_ContainerRelease1].Command;
	HMI_CmdBar_PB[PB_ContainerBlock2].LampON		:= HMI_CmdBar_PB[PB_ContainerBlock2].Command;
	HMI_CmdBar_PB[PB_ContainerBlock2].Blink			:= VAR_ContBlock2.Q1 AND NOT HMI_CmdBar_PB[PB_ContainerBlock2].Command;
	HMI_CmdBar_PB[PB_ContainerRelease2].LampON		:= HMI_CmdBar_PB[PB_ContainerRelease2].Command;
	//HMI_CmdBar_PB[PB_FillerDoorUnlock].LampON		:= OPS.DataOut.HmiFlrDoorUnlock;
	//HMI_CmdBar_PB[PB_SeamerDoorUnlock].LampON		:= OPS.DataOut.HmiSmrDoorUnlock;
END_ACTION
```

#### Command_Bar_PET.st
```iecst
ACTION HMI_CommandBar_Visibility_PET:
	HMI_CmdBar_PB[PB_MixerProcessStart].Visibility		:= CFG_Par.Process.BlendFill;
	HMI_CmdBar_PB[PB_FillerProcessStart].Visibility		:= NOT CFG_Par.Process.BlendFill; //v1.6
	HMI_CmdBar_PB[PB_FillerStartStop].Visibility		:= CFG_Par.Machine.Combi.BF OR CFG_Par.Machine.Combi.BFL OR CFG_Par.Machine.Combi.BLF OR CFG_Par.Machine.Combi.BAF;//V4.A.A.1.6.12
	HMI_CmdBar_PB[PB_ContainerBlock1].Visibility		:= NOT CFG_Par.Machine.Combi.BF AND NOT CFG_Par.Machine.Combi.BFL AND NOT CFG_Par.Machine.Combi.BLF AND NOT CFG_Par.Machine.Combi.BAF;//V4.A.A.1.6.12
	HMI_CmdBar_PB[PB_ContainerRelease1].Visibility		:= NOT CFG_Par.Machine.Combi.BF AND NOT CFG_Par.Machine.Combi.BFL AND NOT CFG_Par.Machine.Combi.BLF AND NOT CFG_Par.Machine.Combi.BAF;//V4.A.A.1.6.12
	HMI_CmdBar_PB[PB_FillerDoorUnlock].Visibility		:= TRUE;
	HMI_CmdBar_PB[PB_FillerLabellerCoupling].Visibility	:= CFG_Par.Machine.Combi.BLF;
	HMI_CmdBar_PB[PB_FillerBlowerCoupling].Visibility	:= CFG_Par.Machine.Combi.BF OR CFG_Par.Machine.Combi.BFL;
	HMI_CmdBar_PB[PB_FillerActisCoupled].Visibility		:= CFG_Par.Machine.Combi.BAF;//V4.A.A.1.6.12
END_ACTION

ACTION HMI_CommandBar_Command_PET:
	VAR_LbrCombiModality(
	SET1	:= EDGEPOS(HMI_CmdBar_PB[PB_FillerLabellerCoupling].ON) AND NOT VAR_LbrCombiModality.Q1,
	RESET	:= EDGEPOS(HMI_CmdBar_PB[PB_FillerLabellerCoupling].ON) AND VAR_LbrCombiModality.Q1
	);

	VAR_BlrCombiModalityReset := FALSE; //V4.A.A.1.6.12h
	IF CFG_Par.Machine.Combi.BF AND NOT OPS.DataOut.FlrModeSelectorAuto THEN //V4.A.A.1.6.12h
		VAR_BlrCombiModalityReset := TRUE;									//V4.A.A.1.6.12h
	END_IF

	//Old Management
	VAR_BlrCombiModality(
	SET1	:= EDGEPOS(HMI_CmdBar_PB[PB_FillerBlowerCoupling].ON) AND NOT VAR_BlrCombiModality.Q1,
	RESET	:= EDGEPOS(HMI_CmdBar_PB[PB_FillerBlowerCoupling].ON) AND VAR_BlrCombiModality.Q1
	);

	//New Management
//	VAR_BlrCombiModality(
//	SET1	:= EDGEPOS(HMI_CmdBar_PB[PB_FillerBlowerCoupling].ON) AND NOT VAR_BlrCombiModality.Q1 AND NOT VAR_BlrCombiModalityReset,//V4.A.A.1.6.12h
//	RESET	:= (EDGEPOS(HMI_CmdBar_PB[PB_FillerBlowerCoupling].ON) AND VAR_BlrCombiModality.Q1) OR VAR_BlrCombiModalityReset,//V4.A.A.1.6.12h
//	);

	VAR_ActCombiModality(//V4.A.A.1.6.12
	SET1	:= EDGEPOS(HMI_CmdBar_PB[PB_FillerActisCoupled].ON) AND NOT VAR_ActCombiModality.Q1,
	RESET	:= EDGEPOS(HMI_CmdBar_PB[PB_FillerActisCoupled].ON) AND VAR_ActCombiModality.Q1
	);

	VAR_ContUnblock1(
	SET1	:= EDGEPOS(HMI_CmdBar_PB[PB_ContainerRelease1].ON) AND NOT VAR_ContUnblock1.Q1,
	RESET	:= (EDGEPOS(HMI_CmdBar_PB[PB_ContainerRelease1].ON) AND VAR_ContUnblock1.Q1) OR EDGEPOS(HMI_CmdBar_PB[PB_ContainerBlock1].ON) OR EDGEPOS(SFT.DataOut.COPInletContConvEmptyRunning)
	);

	VAR_ContBlock1(
	SET1	:= EDGEPOS(HMI_CmdBar_PB[PB_ContainerBlock1].ON) AND NOT VAR_ContBlock1.Q1,
	RESET	:= (EDGEPOS(HMI_CmdBar_PB[PB_ContainerBlock1].ON) AND VAR_ContBlock1.Q1) OR EDGEPOS(HMI_CmdBar_PB[PB_ContainerRelease1].ON)
	);

	HMI_CmdBar_PB[PB_MixerProcessStart].Command			:= BlrFlr.PbMxrProcessCommand OR LbrFlr.PbFlrMixerCommand OR ActFlr.PbFlrMixerCommand;(*V1.61*)(*V4.A.A.1.6.12*)
	HMI_CmdBar_PB[PB_FillerProcessStart].Command		:= HMI_CmdBar_PB[PB_FillerProcessStart].ON		OR BlrFlr.PbFlrProcessCommand OR LbrFlr.PbFlrProcessCommand OR ActFlr.PbFlrProcessCommand;//V4.A.A.1.6.12
	HMI_CmdBar_PB[PB_FillerStartStop].Command			:= HMI_CmdBar_PB[PB_FillerStartStop].ON;
	HMI_CmdBar_PB[PB_ContainerBlock1].Command			:= VAR_ContBlock1.Q1 AND NOT (SFT.DataOut.COPInletContConvEmptyRunning XOR SFT.DataOut.COPInletContConvEmptyDone);
	HMI_CmdBar_PB[PB_ContainerRelease1].Command			:= VAR_ContUnblock1.Q1;;
	HMI_CmdBar_PB[PB_FillerDoorUnlock].Command			:= HMI_CmdBar_PB[PB_FillerDoorUnlock].ON		OR BlrFlr.PbFlrDoorCommand	OR LbrFlr.PbFlrDoorCommand OR ActFlr.PbFlrDoorCommand;//V4.A.A.1.6.12
	HMI_CmdBar_PB[PB_FillerLabellerCoupling].Command	:= VAR_LbrCombiModality.Q1;
	HMI_CmdBar_PB[PB_FillerBlowerCoupling].Command		:= VAR_BlrCombiModality.Q1;
	HMI_CmdBar_PB[PB_FillerActisCoupled].Command		:= VAR_ActCombiModality.Q1;//V4.A.A.1.6.12
END_ACTION

ACTION HMI_CommandBar_Enable_PET:
	HMI_CmdBar_PB[PB_MixerProcessStart].Enable			:= CrbFlr.HMI_ProcessStartEnable;(*V1.61*)
	HMI_CmdBar_PB[PB_FillerProcessStart].Enable			:= SEL(CFG_Par.Process.BlendFill, SkdFlr.HMI_ProcessStartEnable, CrbFlr.HMI_ProcessStartEnable);
	HMI_CmdBar_PB[PB_FillerStartStop].Enable			:= OPS.DataOut.FlrModeSelectorAuto AND NOT AID.DataOut.OneMachineStopAlarm AND//V4.A.A.1.7.0
															(MC_InputOutput.Network.Machine.Status.AutoModalityActive OR MC_InputOutput.Network.Machine.Status.MultiModalityActive) AND NOT FmcFlr.FillingManualTestActive;

	HMI_CmdBar_PB[PB_ContainerBlock1].Enable			:= TRUE;
	HMI_CmdBar_PB[PB_ContainerRelease1].Enable			:= (SFT.DataOut.ManualContainersReleaseEnable OR HMI_CmdBar_PB[PB_ContainerRelease1].Command) AND NOT SFT.DataOut.COPInletContConvEmptyRunning;
	HMI_CmdBar_PB[PB_FillerDoorUnlock].Enable			:= NOT MC_InputOutput.Network.Machine.Status.MachineRunning AND NOT MC_InputOutput.Network.Filler.Status.ModuleRunning AND NOT MC_InputOutput.Network.Inlet.Status.ModuleRunning;
	HMI_CmdBar_PB[PB_FillerLabellerCoupling].Enable		:= LbrFlr.ReadyForCoupling AND LbrFlr.Stopped AND LbrFlr.MachOutFree AND //V1.7.2
															(MNM.DataOut.ReadyForCoupling OR HMI_CmdBar_PB[PB_FillerLabellerCoupling].LampON) AND NOT MC_InputOutput.Network.Machine.Status.MachineRunning; //V4.A.A.1.6.10a
	HMI_CmdBar_PB[PB_FillerBlowerCoupling].Enable		:= BlrFlr.BlrReadyForCoupling AND BlrFlr.Stopped AND
															(MNM.DataOut.ReadyForCoupling OR HMI_CmdBar_PB[PB_FillerBlowerCoupling].LampON) AND NOT MC_InputOutput.Network.Machine.Status.MachineRunning; //V4.A.A.1.6.10a
	HMI_CmdBar_PB[PB_FillerActisCoupled].Enable			:= ActFlr.ReadyForCoupling AND ActFlr.Stopped AND
															(MNM.DataOut.ReadyForCoupling OR HMI_CmdBar_PB[PB_FillerActisCoupled].LampON) AND NOT MC_InputOutput.Network.Machine.Status.MachineRunning;//V4.A.A.1.6.12
	BP_ActisFillingCoupled.Enable						:= HMI_CmdBar_PB[PB_FillerActisCoupled].Enable;//V4.A.A.1.7.0
END_ACTION

ACTION HMI_CommandBar_Status_PET:
	HMI_CmdBar_PB[PB_MixerProcessStart].LampON			:= CrbFlr.HMI_ProcessStartLampOn;(*V1.61*)
	HMI_CmdBar_PB[PB_FillerProcessStart].LampON			:= SEL(CFG_Par.Process.BlendFill, SkdFlr.HMI_ProcessStartLampOn, CrbFlr.HMI_ProcessStartLampOn);
	HMI_CmdBar_PB[PB_ContainerBlock1].Blink				:= VAR_ContBlock1.Q1 AND NOT HMI_CmdBar_PB[PB_ContainerBlock1].Command;
	HMI_CmdBar_PB[PB_ContainerRelease1].LampON			:= HMI_CmdBar_PB[PB_ContainerRelease1].Command;
	HMI_CmdBar_PB[PB_FillerStartStop].LampON 			:= MNM.DataOut.StartLightFixRequest;
	HMI_CmdBar_PB[PB_FillerDoorUnlock].LampON			:= OPS.DataOut.HMIDoorUnlock;
	HMI_CmdBar_PB[PB_FillerLabellerCoupling].LampON		:= HMI_CmdBar_PB[PB_FillerLabellerCoupling].Command;
	HMI_CmdBar_PB[PB_FillerBlowerCoupling].LampON		:= HMI_CmdBar_PB[PB_FillerBlowerCoupling].Command;
	HMI_CmdBar_PB[PB_FillerActisCoupled].LampON			:= HMI_CmdBar_PB[PB_FillerActisCoupled].Command;//V4.A.A.1.6.12
	BP_ActisFillingCoupled.State						:= HMI_CmdBar_PB[PB_FillerActisCoupled].LampON;//V4.A.A.1.7.0

	HMI_CmdBar_PB[PB_FillerStartStop].Blink				:= MNM.DataOut.StartLightBlinkRequest;
	HMI_CmdBar_PB[PB_FillerProcessStart].Blink			:= SEL(CFG_Par.Process.BlendFill, SkdFlr.HMI_ProcessStartBlink, CrbFlr.HMI_ProcessStartBlink);
END_ACTION
```

#### ITC_Mng.st
```iecst
ACTION HMI_ITCMng:
	IF HMI_ITC_Page.PartnerID <> HMI_ITC_PartnerOld OR NOT HMI_ITC_Partner_CFG[HMI_ITC_Page.PartnerID] THEN
		HMI_ITC_Page.PartnerID	:= LIMIT(CST_MinITCPartner, HMI_ITC_Page.PartnerID, CST_MaxITCPartner);
		FOR VAR_ITCindex := HMI_ITC_Page.PartnerID TO CST_MaxITCPartner DO
			IF HMI_ITC_Partner_CFG[VAR_ITCindex] THEN
				HMI_ITC_Page.PartnerID := VAR_ITCindex;
				EXIT;
			END_IF
		END_FOR

		HMI_ITC_Page.PageNum	:= 0;
		HMI_ITC_PartnerOld		:= HMI_ITC_Page.PartnerID;
		HMI_ITC_PageData.PageUp.Enable		:= FALSE;
		HMI_ITC_PageData.PageDown.Enable	:= FALSE;
	END_IF

	HMI_ITC_PageData ACCESS (ADR(HMI_ITC_PageDB[CST_MinITCPartner]) + MIN(HMI_ITC_Page.PartnerID - CST_MinITCPartner, CST_MaxITCPartner) * SIZEOF(HMI_ITC_PageDB[CST_MinITCPartner]));

	HMI_ITC_PageData.PageUp.LampON		:= HMI_ITC_PageData.PageUp.ON AND HMI_ITC_PageData.PageUp.Enable;
	HMI_ITC_PageData.PageDown.LampON	:= HMI_ITC_PageData.PageDown.ON AND HMI_ITC_PageData.PageDown.Enable;

	IF EDGEPOS(HMI_ITC_PageData.PageUp.LampON) THEN
		HMI_ITC_Page.PageNum	:= LIMIT(0, HMI_ITC_Page.PageNum + 1, 20);
		HMI_ITC_PageData.PageUp.Enable		:= FALSE;
		HMI_ITC_PageData.PageDown.Enable	:= FALSE;
	END_IF

	IF EDGEPOS(HMI_ITC_PageData.PageDown.LampON) THEN
		HMI_ITC_Page.PageNum	:= LIMIT(0, HMI_ITC_Page.PageNum - 1, 20);
		HMI_ITC_PageData.PageDown.Enable	:= FALSE;
		HMI_ITC_PageData.PageUp.Enable		:= FALSE;
	END_IF
END_ACTION
```

#### Counter_Mng.st
```iecst
ACTION HMI_CounterInit:
	HMI_CounterCfgPartial.MachineCounters.HmiData[FillerLaps].Description				:= '@CounterDescription_001';
	HMI_CounterCfgPartial.MachineCounters.HmiData[ClosingUnit1Laps].Description			:= '@CounterDescription_002';
	HMI_CounterCfgPartial.MachineCounters.HmiData[ClosingUnit2Laps].Description			:= '@CounterDescription_003';
	HMI_CounterCfgPartial.MachineCounters.HmiData[RinserLaps].Description				:= '@CounterDescription_004';
	HMI_CounterCfgPartial.MachineCounters.HmiData[FlaworDoserLaps].Description			:= '@CounterDescription_005';
	HMI_CounterCfgPartial.MachineCounters.HmiData[PulpDoserLaps].Description			:= '@CounterDescription_006';
	HMI_CounterCfgPartial.MachineCounters.HmiData[PowerOn].Description					:= '@CounterDescription_007';
	HMI_CounterCfgPartial.MachineCounters.HmiData[RotatingTime].Description				:= '@CounterDescription_048'; //V1.7.4

	HMI_CounterCfgPartial.ContainersCounters.HmiData[FillingFault].Description			:= '@CounterDescription_008';
	HMI_CounterCfgPartial.ContainersCounters.HmiData[FillingBurst].Description			:= '@CounterDescription_009';
	HMI_CounterCfgPartial.ContainersCounters.HmiData[ClosingUnit1Fault].Description		:= '@CounterDescription_010';
	HMI_CounterCfgPartial.ContainersCounters.HmiData[ClosingUnit2Fault].Description		:= '@CounterDescription_011';
	HMI_CounterCfgPartial.ContainersCounters.HmiData[RinsingFault].Description			:= '@CounterDescription_012';
	HMI_CounterCfgPartial.ContainersCounters.HmiData[PulpDoserFault].Description		:= '@CounterDescription_013';
	HMI_CounterCfgPartial.ContainersCounters.HmiData[FlaworDoserFault].Description		:= '@CounterDescription_014';
	HMI_CounterCfgPartial.ContainersCounters.HmiData[BurstEjected].Description			:= '@CounterDescription_015';
	HMI_CounterCfgPartial.ContainersCounters.HmiData[ManualEjected].Description			:= '@CounterDescription_016';
	HMI_CounterCfgPartial.ContainersCounters.HmiData[LowFillingEjected].Description		:= '@CounterDescription_017';
	HMI_CounterCfgPartial.ContainersCounters.HmiData[NotFilledEjected].Description		:= '@CounterDescription_018';
	HMI_CounterCfgPartial.ContainersCounters.HmiData[ContainersEntered].Description		:= '@CounterDescription_019';
	HMI_CounterCfgPartial.ContainersCounters.HmiData[ContainersProduced].Description	:= '@CounterDescription_020';
	HMI_CounterCfgPartial.ContainersCounters.HmiData[EjectionBySIS].Description			:= '@CounterDescription_045'; //V4.A.A.1.6.8
	HMI_CounterCfgPartial.ContainersCounters.HmiData[BottleProduceToCvo].Description;//			 := '@CounterDescription_046'; //V4.A.A.1.6.8
	HMI_CounterCfgPartial.ContainersCounters.HmiData[Spare].Description;// := '@CounterDescription_047'; //V4.A.A.1.6.8

	HMI_CounterCfgPartial.ProcessCounters.HmiData[FillerProduction].Description			:= '@CounterDescription_021';
	HMI_CounterCfgPartial.ProcessCounters.HmiData[ClosingUnit1Production].Description	:= '@CounterDescription_022';
	HMI_CounterCfgPartial.ProcessCounters.HmiData[ClosingUnit2Production].Description	:= '@CounterDescription_023';
	HMI_CounterCfgPartial.ProcessCounters.HmiData[RinserProduction].Description			:= '@CounterDescription_024';
	HMI_CounterCfgPartial.ProcessCounters.HmiData[PulpDoserProduction].Description		:= '@CounterDescription_025';
	HMI_CounterCfgPartial.ProcessCounters.HmiData[FlaworDoserProduction].Description	:= '@CounterDescription_026';
	HMI_CounterCfgPartial.ProcessCounters.HmiData[Cop].Description						:= '@CounterDescription_027';
	HMI_CounterCfgPartial.ProcessCounters.HmiData[FillerCip].Description				:= '@CounterDescription_044';
	HMI_CounterCfgPartial.ProcessCounters.HmiData[ClosingUnit1Cip].Description			:= '@CounterDescription_028';
	HMI_CounterCfgPartial.ProcessCounters.HmiData[ClosingUnit2Cip].Description			:= '@CounterDescription_029';
	HMI_CounterCfgPartial.ProcessCounters.HmiData[RinserCip].Description				:= '@CounterDescription_030';
	HMI_CounterCfgPartial.ProcessCounters.HmiData[PulpDoserCip].Description				:= '@CounterDescription_031';
	HMI_CounterCfgPartial.ProcessCounters.HmiData[FlaworDoserCip].Description			:= '@CounterDescription_032';

	HMI_CounterCfgPartial.EcoCounters.HmiData[Power].Description						:= '@CounterDescription_033';
	HMI_CounterCfgPartial.EcoCounters.HmiData[Air].Description							:= '@CounterDescription_034';
	HMI_CounterCfgPartial.EcoCounters.HmiData[GeneralCO2].Description					:= '@CounterDescription_035';
	HMI_CounterCfgPartial.EcoCounters.HmiData[ClosingUnitCO2].Description				:= '@CounterDescription_036';
	HMI_CounterCfgPartial.EcoCounters.HmiData[N2].Description							:= '@CounterDescription_037';
	HMI_CounterCfgPartial.EcoCounters.HmiData[ProcessWater].Description					:= '@CounterDescription_038';
	HMI_CounterCfgPartial.EcoCounters.HmiData[CopWater].Description						:= '@CounterDescription_039';
	HMI_CounterCfgPartial.EcoCounters.HmiData[BottomBottleCoolingWater].Description		:= '@CounterDescription_040';
	HMI_CounterCfgPartial.EcoCounters.HmiData[Product].Description						:= '@CounterDescription_041';
	HMI_CounterCfgPartial.EcoCounters.HmiData[Steam].Description						:= '@CounterDescription_042';
	HMI_CounterCfgPartial.EcoCounters.HmiData[FoodSteam].Description					:= '@CounterDescription_043';
	HMI_CounterCfgPartial.EcoCounters.HmiData[ProductWater].Description					:= '@CounterDescription_049'; //V4.A.A.1.6.14k
	HMI_CounterCfgPartial.EcoCounters.HmiData[Syrup].Description						:= '@CounterDescription_050'; //V4.A.A.1.6.14k

	HMI_CounterCfgPartial.EcoCounters.HmiData[Power].Unit								:= '';
	HMI_CounterCfgPartial.EcoCounters.HmiData[Air].Unit									:= '';
	HMI_CounterCfgPartial.EcoCounters.HmiData[GeneralCO2].Unit							:= '';
	HMI_CounterCfgPartial.EcoCounters.HmiData[ClosingUnitCO2].Unit						:= '';
	HMI_CounterCfgPartial.EcoCounters.HmiData[N2].Unit									:= '';
	HMI_CounterCfgPartial.EcoCounters.HmiData[ProcessWater].Unit						:= '';
	HMI_CounterCfgPartial.EcoCounters.HmiData[CopWater].Unit							:= '';
	HMI_CounterCfgPartial.EcoCounters.HmiData[BottomBottleCoolingWater].Unit			:= '';
	HMI_CounterCfgPartial.EcoCounters.HmiData[Product].Unit								:= '';
	HMI_CounterCfgPartial.EcoCounters.HmiData[Steam].Unit								:= '';
	HMI_CounterCfgPartial.EcoCounters.HmiData[FoodSteam].Unit							:= '';
	HMI_CounterCfgPartial.EcoCounters.HmiData[ProductWater].Unit						:= ''; //V4.A.A.1.6.14k
	HMI_CounterCfgPartial.EcoCounters.HmiData[Syrup].Unit								:= ''; //V4.A.A.1.6.14k
END_ACTION

ACTION HMI_CounterMng:
	CASE HMI_CounterPageCategory OF
		0:
			HMI_CounterPartialCfgPageDB		ACCESS	(ADR(HMI_CounterCfgPartial.MachineCounters));
			HMI_CounterPartialDataPageDB	ACCESS	(ADR(HMI_CounterDataPartial.MachineCounters));
			HMI_CounterTotalCfgPageDB		ACCESS	(ADR(HMI_CounterCfgTotal.MachineCounters));
			HMI_CounterTotalDataPageDB		ACCESS	(ADR(HMI_CounterDataTotal.MachineCounters));

		10:
			HMI_CounterPartialCfgPageDB		ACCESS	(ADR(HMI_CounterCfgPartial.ContainersCounters));
			HMI_CounterPartialDataPageDB	ACCESS	(ADR(HMI_CounterDataPartial.ContainersCounters));
			HMI_CounterTotalCfgPageDB		ACCESS	(ADR(HMI_CounterCfgTotal.ContainersCounters));
			HMI_CounterTotalDataPageDB		ACCESS	(ADR(HMI_CounterDataTotal.ContainersCounters));

		20:
			HMI_CounterPartialCfgPageDB		ACCESS	(ADR(HMI_CounterCfgPartial.ProcessCounters));
			HMI_CounterPartialDataPageDB	ACCESS	(ADR(HMI_CounterDataPartial.ProcessCounters));
			HMI_CounterTotalCfgPageDB		ACCESS	(ADR(HMI_CounterCfgTotal.ProcessCounters));
			HMI_CounterTotalDataPageDB		ACCESS	(ADR(HMI_CounterDataTotal.ProcessCounters));

		30:
			HMI_CounterPartialCfgPageDB		ACCESS	(ADR(HMI_CounterCfgPartial.EcoCounters));
			HMI_CounterPartialDataPageDB	ACCESS	(ADR(HMI_CounterDataPartial.EcoCounters));
			HMI_CounterTotalCfgPageDB		ACCESS	(ADR(HMI_CounterCfgTotal.EcoCounters));
			HMI_CounterTotalDataPageDB		ACCESS	(ADR(HMI_CounterDataTotal.EcoCounters));
	END_CASE

	HMI_TotalBottleProduced	:= HMI_CounterDataTotal.ContainersCounters.CounterData[ContainersProduced].CounterValue;

	//DATA TO EXCHANGE IN HMI WITH BLOWER //V4.A.A.1.7.0
	HMI_CounterHome.SS2P.Visibility 	:= FALSE;//not used in Glass Machine
	HMI_CounterHome.SS2P.Enable			:= FALSE;//not used in Glass Machine
	HMI_CounterHome.SS2P.LampON 		:= HMI_CounterHome.SS2P.ON;
//	HMI_CounterHome.CounterValue[0] 	:= MAX(0,HMI_CounterDataPartial.ContainersCounters.CounterData[SIS_ContainersProducedToBlower].CounterValue -
//												HMI_CounterDataPartial.ContainersCounters.CounterData[SIS_EjectionToBlower].CounterValue);
//	HMI_CounterHome.CounterValue[1]		:= HMI_CounterDataPartial.ContainersCounters.CounterData[SIS_EjectionToBlower].CounterValue;

END_ACTION
```

#### HMI_Init_CFG.st
```iecst
PROGRAM _INIT
	//AID
	HMI_AID_Loading;

	//ALR - Alarm
	HMI_ALR_Loading;

	//CAP - Capper
	HMI_CAP_Loading;

	//CRW - Crowner
	HMI_CRW_Loading;

	// CO - Change Over
	HMI_CO_Loading;

	//COP - Cleaning out place
	HMI_COP_Loading;

	//CSR - Container Size Regulation
	HMI_CSR_Loading;

	//DMC - Dummy containers
	HMI_DMC_Loading;

	//GNS - General safety
	HMI_GNS_Loading;

	//MAU - Machine auxiliary
	HMI_MAU_Loading;

	//MNM - Main drive
	HMI_MNM_Loading;

	//MNT - Maintenance
	HMI_MNT_Loading;

	//ICO - Intelli Change Over
	HMI_ICO_Loading;

	//ITC - Interchange
	HMI_ITC_Loading;

	//OPS - Operator safety
	HMI_OPS_Loading;

	//HMI - Option Page
	HMI_OPT_Loading;

	//PAO - HMI PAO Page
	HMI_PAO_Loading;

	//RNS - RINSER
	HMI_RNS_Loading;

	//SFT - SHIFT REGISTER
	HMI_SFT_Loading;

	//TNK - Tank
	HMI_TNK_Loading;

	//DAQ - Data Aquisition v1.7.4a
	HMI_DAQ_Loading;

	//Device (Valves - Instruments - Pumps)
	HMI_Valves_Loading;
	HMI_Instruments_Loading;
	HMI_Pumps_Loading;

	//HMI Variables
	HMI_Variables_Loading;

	HMI_CounterInit;

	//CTP - CAP TRATMENT PREPARATION
	HMI_CTP_Loading;

	//DOS - PULPDOSER v999hema
	HMI_DOS_Loading;

END_PROGRAM
```

### Package Logical/02_HMI/HMI_Types - HMI Global data types

### HMI_CAP.typ
```iecst
TYPE
	HMI_CAP_ManualCapsSelection_Type : 	STRUCT
		Value : USINT;
		Visibility : BOOL;
	END_STRUCT;
	HMI_CAP_ConfigStructure_Type : 	STRUCT
		Caps : CFG_Cap_Par_Type;
		CfgPresence : HMI_CAP_ConfigStructPres_Type;
		SavePB : PB_Type;
		LoadPB : PB_Type;
	END_STRUCT;
	HMI_CAP_ConfigStructPres_Type : 	STRUCT
		Channel : BOOL;
		BufferPresent : BOOL;
		BufferSize : BOOL;
		CamHeight : BOOL;
		HeadRotation : BOOL;
		PaP : BOOL;
	END_STRUCT;
	HMI_CAP_State_Type : 	STRUCT
		Sequencer : Seq_Type; (*Step Actual*)
		Signals : Signals_Type;
	END_STRUCT;
	HMI_CAP_Greasing_Type : 	STRUCT
		Cycle_Number : UINT;
		Cycle_Request_H : UINT;
		Cycle_TimeOut : UDINT;
		Turret_Cycle_Number : UINT;
		Cycle_RunningTime : UINT;
		Cycle_PauseTime : UDINT;
		Cycle_Running : BOOL;
		Cycle_Alarm : BOOL;
		Pump_Running : BOOL;
	END_STRUCT;
	HMI_CAP_SikoMotor_Type : 	STRUCT  (*V1.61*)
		MotorMax : UINT; (*Head Configuration Number*)
		Data : HMI_CAP_SikoData_Type; (*Data Report Page*)
		Maintenance : ARRAY[0..10]OF Info_Type; (*Maintenance Area*)
		Calibration : HMI_CAP_SikoCal_Type; (*Calibration Area*)
		PageUp : PB_Type := (0); (*Head Scroll in Data Report Page*)
		PageDown : PB_Type := (0); (*Head Scroll in Data Report Page*)
	END_STRUCT;
	HMI_CAP_Brush_Type : 	STRUCT  (*v1.4*)
		HeadMax : UINT; (*Head Configuration Number*)
		Data : HMI_CAP_Data_Type; (*Data Report Page*)
		Maintenance : ARRAY[0..10]OF Info_Type; (*Maintenance Area*)
		Calibration : HMI_CAP_Cal_Type; (*Calibration Area*)
		PageUp : PB_Type := (0); (*Head Scroll in Data Report Page*)
		PageDown : PB_Type := (0); (*Head Scroll in Data Report Page*)
		MaintenanceReadWrite : SS2P_Type; (*//V4.A.A.1.6.11*)
	END_STRUCT;
	HMI_CAP_SikoData_Type : 	STRUCT  (*V1.61*)
		Motor : HMI_CAP_SikoMotorData_Type; (*Data Report*)
		MotorStatus : HMI_CAP_Status_Type; (*Boolean Head Status (Zalkin Only)*)
	END_STRUCT;
	HMI_CAP_Data_Type : 	STRUCT  (*v1.4*)
		HeadNr : UINT; (*Head Request for Diagnostic*)
		Head : ARRAY[0..15]OF HMI_CAP_Head_Type; (*Data Report*)
		HeadStatus : HMI_CAP_Status_Type; (*Boolean Head Status (Zalkin Only)*)
	END_STRUCT;
	HMI_CAP_SikoMotorData_Type : 	STRUCT  (*V1.61*)
		MotorNr : USINT;
		PowerOk : BOOL;
		Enabled : BOOL;
		Ready : BOOL;
		Running : BOOL;
		InPosition : BOOL;
		Error : BOOL;
		BatteryWarning : BOOL;
		xParamRwBusy : BOOL; (*Parameter read/write operation is busy*)
		xParamRwError : BOOL; (*Parameter read/write operation is in error*)
		xParamRwDone : BOOL; (*Parameter read/write operation is done*)
		wPositionVelocity : UINT; (*Jog velocity*)
		wJogVelocity : UINT; (*Current limit*)
		bCurrentLimit : USINT; (*Sense of rotation*)
		bSenseOfRotation : USINT;
	END_STRUCT;
	HMI_CAP_Head_Type : 	STRUCT  (*v1.4*)
		HeadNr : UINT; (*Head Displayed on Row*)
		Data1 : UINT; (*//In arol Equatorque is value of Heads Torque*)
		Data2 : UINT;
		Totalizer00 : UINT;
		Totalizer01 : UINT;
		Totalizer02 : UINT;
		Totalizer03 : UINT;
		Totalizer04 : UINT;
		Totalizer05 : UINT;
		Totalizer06 : UINT;
		Totalizer07 : UINT;
		Bool00 : BOOL; (*//In arol Equatorque RejectionSignal*)
		Bool01 : BOOL; (*//In arol Equatorque NoLoad*)
		Bool02 : BOOL; (*//In arol Equatorque NoClosure*)
		Bool03 : BOOL; (*//In arol Equatorque InTorque*)
		Bool04 : BOOL; (*//In arol Equatorque BadClosure*)
		Bool05 : BOOL; (*//In arol Equatorque FollowingError*)
		Bool06 : BOOL; (*//In arol Equatorque BadClosure*)
		Bool07 : BOOL; (*//In arol Equatorque NoUnwrap*)
		LineVisibility : BOOL;
	END_STRUCT;
	HMI_CAP_Cal_Type : 	STRUCT  (*v1.4*)
		HeadNr : UINT; (*Head Request for Calibration*)
		HeadUp : PB_Type := (0); (*Head Scroll in Calibration Page*)
		HeadDown : PB_Type := (0); (*Head Scroll in Calibration Page*)
		Sequence : SeqTextBar_Type; (*Calibration Sequencer Status*)
		Data : ARRAY[0..14]OF Info_Type; (*//V4.A.A.1.6.12*)
		HeadStatus : HMI_CAP_Status_Type; (*Boolean Head Status (Zalkin Only)*)
		SequencerPerc : INT; (*AROL Equatorque Calibration -Sequencer Step Percentage Display V4.A.A.1.6.12*)
	END_STRUCT;
	HMI_CAP_SikoCal_Type : 	STRUCT  (*V1.61*)
		MotorNr : UINT; (*Motor Siko Request for Calibration*)
		MotorForward : PB_Type := (0); (*Move Motor Forward in Jog Mode*)
		MotorStartPositioning : PB_Type := (0); (*Motor Move to Target Position*)
		MotorBackward : PB_Type := (0); (*Move Motor Backward in Jog Mode*)
		MotorWriteParameter : PB_Type; (*Write Parameter*)
		MotorReadParameter : PB_Type; (*Read Parameter*)
		MotorHoming : PB_Type; (*Homing Motor*)
		Sequence : SeqTextBar_Type; (*Calibration Sequencer Status*)
		Data : Info_Type;
	END_STRUCT;
	HMI_CAP_Status_Type : 	STRUCT  (*v1.4*)
		Visibility : ARRAY[0..7]OF BOOL;
		Status : ARRAY[0..7]OF BOOL;
	END_STRUCT;
	HMI_CAP_DataCfg_Type : 	STRUCT  (*v1.4*)
		Present : BOOL;
		Name : STRING[40];
	END_STRUCT;
	HMI_CAP_ZoneCfg_Type : 	STRUCT  (*v1.5*)
		Present : BOOL;
		Name : STRING[8];
	END_STRUCT;
	HMI_CAP_BufferAdjust_Type : 	STRUCT  (*//V4.A.A.1.6.11*)
		Position_Actual : REAL;
		Position_Request : REAL;
	END_STRUCT;
	HMI_CAP_HRM_Type : 	STRUCT  (*//V4.A.A.1.6.11*)
		ProdSpeedRPM : UINT;
		HeadSpeedRPM : UINT;
		DiagCode : UINT;
		ActualCurrent : DINT; (*v1.7.4*)
		ProdSpeedBPH : REAL;
	END_STRUCT;
END_TYPE
```

### HMI_CFG.typ
```iecst
TYPE
	HMI_PAO_Type : 	STRUCT
		FirstConfigLoaded : BOOL;
		Saved : BOOL;
		Loaded : BOOL;
		Busy : BOOL;
		ErrorLoading : BOOL;
		ErrorSaving : BOOL;
	END_STRUCT;
	HMI_CFG_Display_Type : 	STRUCT
		Name : STRING[100];
		Visibility : BOOL;
		ValueR : REAL;
		PresentR : BOOL;
		ValueB : BOOL;
		PresentB : BOOL;
		ValueI : DINT;
		PresentI : BOOL;
		ValueSt : STRING[100];
		PresentSt : BOOL;
	END_STRUCT;
END_TYPE
```

### HMI_CO.typ
```iecst
TYPE
	HMI_APCO_Type : 	STRUCT
		Action : HMI_APCO_Action_Type;
		Recipe : HMI_APCO_Recipe_Type;
	END_STRUCT;
	HMI_APCO_Recipe_Type : 	STRUCT
		ProductTypeActual : UINT;
		ProductTypeNext : UINT;
	END_STRUCT;
	HMI_APCO_Recipe_Download_Type : 	STRUCT
		Request : BOOL;
		Ended : BOOL;
	END_STRUCT;
	HMI_APCO_Action_Type : 	STRUCT
		CheckPoints : ARRAY[0..15]OF HMI_APCO_Action_CheckPoints_Type;
		TypeOfChange : INT; (*V4.A.A.1.6.12*)
		CheckPointActive : INT; (*V4.A.A.1.6.12*)
	END_STRUCT;
	HMI_APCO_Action_CheckPoints_Type : 	STRUCT
		Visibility : BOOL;
		IndexText : UINT;
		ON : BOOL;
	END_STRUCT;
END_TYPE
```

### HMI_CRW.typ
```iecst
TYPE
	HMI_CRW_ManualCrwSelection_Type : 	STRUCT
		Value : USINT;
		Visibility : BOOL;
	END_STRUCT;
	HMI_CRW_ConfigStructure_Type : 	STRUCT
		Crown : CFG_Crw_Par_Type;
		Presence : HMI_CRW_ConfigStructPres_Type;
		SavePB : PB_Type;
		LoadPB : PB_Type;
	END_STRUCT;
	HMI_CRW_ConfigStructPres_Type : 	STRUCT
		Channel : BOOL;
	END_STRUCT;
END_TYPE
```

### HMI_CSR.typ
```iecst
TYPE
	HMI_CSR_Data_Type : 	STRUCT
		TnkPositionPv : REAL;
		TnkPositionSp : REAL;
		ColumnPositionPv : REAL;
		ColumnPositionSp : REAL;
		RnsPositionSp : REAL;
		RnsPositionPv : REAL;
		CapPositionSp : REAL;
		CapPositionPv : REAL;
		CrwPositionSp : REAL;
		CrwPositionPv : REAL;
		RcpMaxValue : REAL;
		RcpMinValue : REAL;
		CrwPageVisibility : BOOL;
		CapPageVisibility : BOOL;
		FillerAlarmActive : BOOL;
		CrownerAlarmActive : BOOL;
		CapperAlarmActive : BOOL;
		RinserAlarmActive : BOOL;
	END_STRUCT;
	HMI_CSR_SikoMotorData_Type : 	STRUCT  (* *) (* *) (*13*)
		ActualPosition : REAL; (* *) (* *) (*14*)
		PR_AccelerationSpeed : INT; (* *) (* *) (*15*)
		PR_CalibrationValue : REAL; (* *) (* *) (*16*)
		PR_Delta_Inch : DINT; (* *) (* *) (*17*)
		PR_GearIn : INT; (* *) (* *) (*18*)
		PR_GearOut : INT; (* *) (* *) (*19*)
		PR_JogSpeed : INT; (* *) (* *) (*20*)
		PR_KP : INT; (* *) (* *) (*21*)
		PR_TD : INT; (* *) (* *) (*22*)
		PR_TI : INT; (* *) (* *) (*23*)
		PR_Upper_Limit : REAL; (* *) (* *) (*24*)
		PR_Lower_Limit : REAL; (* *) (* *) (*25*)
		PR_PositionSpeed : INT; (* *) (* *) (*26*)
		PR_PosWindows : INT; (* *) (* *) (*27*)
		PR_RotationSense : INT; (* *) (* *) (*28*)
		PR_Spindle_Pitch : INT; (* *) (* *) (*29*)
		PR_SystemStatus : INT; (* *) (* *) (*30*)
		Status : UINT; (* *) (* *) (*31*)
	END_STRUCT;
	HMI_CSR_SikoActualPosition_Type : 	STRUCT  (* *) (* *) (*33*)
		OutConveyor_Guide : INT; (* *) (* *) (*34*)
		OutConveyor_Height : INT; (* *) (* *) (*35*)
		Position_Actual : REAL; (* *) (* *) (*36*)
		Position_Request : REAL; (* *) (* *) (*37*)
		PositionGuide_Actual : REAL; (*v1.5*) (* *) (*36*)
		PositionGuide_Request : REAL; (*v1.5*) (* *) (*37*)
	END_STRUCT;
END_TYPE
```

### HMI_COP.typ
```iecst
TYPE
	HMI_COP_StatusWidget_Type : 	STRUCT
		Running : BOOL;
		RemaningTime : DINT;
		Mode : INT; (*0: Idle
1: Rinse
2: Rinse hot
3: Wait
4: Foam 1
5: Foam 2
6: Foam 3
10: High speed
11: Emptying with air (purge)
20: Manual*)
	END_STRUCT;
	HMI_COP_ZoneCfg_Type : 	STRUCT
		Present : BOOL;
		Name : STRING[15];
	END_STRUCT;
	HMI_COP_Rcp_Type : 	STRUCT
		Phase : ARRAY[0..CST_COP_PhaseMaxNr]OF HMI_COP_RcpPhase_Type;
	END_STRUCT;
	HMI_COP_RcpSelection_Type : 	STRUCT
		ConfigPresent : BOOL;
		Selected : BOOL;
		Enable : BOOL := TRUE;
		Name : STRING[150];
	END_STRUCT;
	HMI_COP_RcpPhase_Type : 	STRUCT
		PhaseType : USINT;
		Time_SP : UINT;
		PumpPressure_SP : REAL;
		WaterPressure_SP : REAL;
		AirPressure_SP : REAL;
		ValveOpening_SP : REAL;
		Custom01 : REAL;
		Valves_Configuration : UDINT;
	END_STRUCT;
	HMI_COP_RcpInfo_Type : 	STRUCT
		Rcp : HMI_COP_RcpInfoRcp_Type;
		Phase : HMI_COP_RcpInfoPhase_Type;
	END_STRUCT;
	HMI_COP_RcpInfoRcp_Type : 	STRUCT
		Name : STRING[150];
		PhaseNr : USINT;
		TimeAct : UDINT;
		TimePreset : UDINT;
		TimeRemaining : UDINT;
	END_STRUCT;
	HMI_COP_RcpInfoPhase_Type : 	STRUCT
		Nr : USINT;
		Type : USINT;
		TimeAct : UDINT;
		TimePreset : UDINT;
		TimeRemaining : UDINT;
	END_STRUCT;
	HMI_COP_State_Type : 	STRUCT
		Sequencer : Seq_Type; (*Step Actual*)
		Signals : Signals_Type;
	END_STRUCT;
	HMI_COP_ITC_Type : 	STRUCT
		In : HMI_COP_ITC_In_Type;
		Out : HMI_COP_ITC_Out_Type;
	END_STRUCT;
	HMI_COP_ITC_In_Type : 	STRUCT
		CycleActive : BOOL;
		CycleEnded : BOOL;
		Alarm : BOOL;
	END_STRUCT;
	HMI_COP_ITC_Out_Type : 	STRUCT
		ReadyForFoaming : BOOL;
		Alarm : BOOL;
	END_STRUCT;
END_TYPE
```

### HMI_GNS.typ
```iecst
(*LAMP TEST*)

TYPE
	HMI_Beacon_Type : 	STRUCT
		LightGreen : HMI_BeaconLamp_Type;
		LightBlue : HMI_BeaconLamp_Type;
		LightYellow : HMI_BeaconLamp_Type;
		LightRed : HMI_BeaconLamp_Type;
		LightWhite : HMI_BeaconLamp_Type;
		Horn : HMI_BeaconLamp_Type;
	END_STRUCT;
	HMI_BeaconLamp_Type : 	STRUCT
		Present : BOOL;
		ON : BOOL;
		Blink : BOOL;
	END_STRUCT;
	HMI_BeaconHome_Type : 	STRUCT
		Present : BOOL;
		LightGreen : HMI_BeaconLamp_Type;
		LightBlue : HMI_BeaconLamp_Type;
		LightYellow : HMI_BeaconLamp_Type;
		LightRed : HMI_BeaconLamp_Type;
		LightWhite : HMI_BeaconLamp_Type;
		Horn : HMI_BeaconLamp_Type;
	END_STRUCT;
END_TYPE
```
